// TwinCAT 3 PLC project Main
// ProgramVersion: 3.1.4023.0
// libraries:
//   Tc2_Standard, * (Beckhoff Automation GmbH)
//   Tc2_System, * (Beckhoff Automation GmbH)
//   Tc3_Module, * (Beckhoff Automation GmbH)
//   TcUnit, * (www.tcunit.org)
//   mobject-constants-datatype-limits,1.0.0,mobject
//   mobject-deserialization,0.3.0,mobject
//   mobject-errors,0.3.0,mobject
//   mobject-json,1.6.0,mobject
//   mobject-serialization,0.5.0,mobject
// project tree:
//   / PlcTask.TcTTO
//   POUs/ MAIN.TcPOU
//   Tests/ JsonDeserializerArrayForwardEnumerator_TestSuite.TcPOU, JsonDeserializerObjectForwardEnumerator_TestSuite.TcPOU, JsonDomParser_TestSuite.TcPOU, JsonSerializer_TestSuite.TcPOU, JsonDeserializer_TestSuite.TcPOU
//   Tests/Mocks/ MockSerializableUserObject.TcPOU, MockDeserializableUserObject.TcPOU, MockSerializableArray.TcPOU
// real-time tasks:
//   TASK PlcTask: cycle T#10ms, priority 20, ADS port 350

CONFIGURATION Main
    RESOURCE PLC ON TwinCAT3
        TASK PlcTask(INTERVAL := T#10ms, PRIORITY := 20);
        PROGRAM MAIN WITH PlcTask : MAIN;
    END_RESOURCE
END_CONFIGURATION

// ---- POUs/MAIN.TcPOU
PROGRAM MAIN
VAR
	jsonDomParser_TestSuite : JsonDomParser_TestSuite;
	jsonSerializer_TestSuite : JsonSerializer_TestSuite;
	jsonDeserializer_TestSuite : JsonDeserializer_TestSuite;
	jsonDeserializerArrayForwardEnumerator_TestSuite : JsonDeserializerArrayForwardEnumerator_TestSuite;
	jsonDeserializerObjectForwardEnumerator_TestSuite : JsonDeserializerObjectForwardEnumerator_TestSuite;
END_VAR

TcUnit.RUN();

END_PROGRAM

// ---- Tests/JsonDomParser_TestSuite.TcPOU
FUNCTION_BLOCK JsonDomParser_TestSuite EXTENDS TcUnit.FB_TestSuite
VAR
	jsonParser : JsonDomParser;
END_VAR

ModifyBoolArrayMemberFromJsonString();
ModifyDIntArrayMemberFromJsonString();
ModifyDIntPropertyFromJsonString();
ModifyFalseBoolPropertyFromJsonString();
ModifyIntArrayMemberFromJsonString();
ModifyIntPropertyFromJsonString();
ModifyLRealArrayMemberFromJsonString();
ModifyLRealPropertyFromJsonString();
ModifyRealArrayMemberFromJsonString();
ModifyRealPropertyFromJsonString();
ModifyStringPropertyFromJsonString();
ModifyTrueBoolPropertyFromJsonString();
ModifyUDIntArrayMemberFromJsonString();
ModifyUDIntPropertyFromJsonString();
ModifyValueFromChainedProperty();
ReadBoolArrayMemberFromJsonString();
ReadDIntArrayMemberFromJsonString();
ReadDIntPropertyFromJsonString();
ReadFalseBoolPropertyFromJsonString();
ReadIntArrayMemberFromJsonString();
ReadIntPropertyFromJsonString();
ReadLRealArrayMemberFromJsonString();
ReadLRealPropertyFromJsonString();
ReadRealArrayMemberFromJsonString();
ReadRealPropertyFromJsonString();
ReadStringPropertyFromJsonString();
ReadTrueBoolPropertyFromJsonString();
ReadUDIntArrayMemberFromJsonString();
ReadUDIntPropertyFromJsonString();
ReadValueFromChainedProperties();
TestTryLocateMethod();
TestTryWriteBoolMethod();
TestTryWriteDintMethod();
TestTryWriteIntMethod();
TestTryWriteLRealMethod();
TestTryWriteRealMethod();
TestTryWriteStringMethod();
TestTryWriteUdintMethod();

METHOD PUBLIC ModifyBoolArrayMemberFromJsonString
VAR_INPUT
END_VAR
VAR
	jsonTestString : T_MAXSTRING := '{"myArray" : [false, false, false]}';
	newValue : BOOL := TRUE;
	modifyResult : BOOL;
	result : BOOL;
	readResult : BOOL;
END_VAR
TEST('ModifyBoolArrayMemberFromJsonString');

// @TEST-RUN
jsonParser.ParseDocument(jsonTestString);
modifyResult := jsonParser.TryModify('.myArray[1]',newValue);
readResult := jsonParser.TryRead('.myArray[1]',result);
jsonParser.NewDocument();

// @TEST-ASSERT
AssertTrue(Condition := result, Message := 'Did not modify to the correct value');
AssertTrue(Condition := readResult, Message := 'Did not report a modify was successful');

TEST_FINISHED();
END_METHOD

METHOD PUBLIC ModifyDIntArrayMemberFromJsonString
VAR_INPUT
END_VAR
VAR
	jsonTestString : T_MAXSTRING := '{"myArray" : [123,456,789]}';
	newValue : DINT := 654;
	modifyResult : BOOL;
	actual : DINT;
	expected : DINT := 654;
	readResult : BOOL;
END_VAR
TEST('ModifyDIntArrayMemberFromJsonString');

// @TEST-RUN
jsonParser.ParseDocument(jsonTestString);
modifyResult := jsonParser.TryModify('.myArray[1]',newValue);
readResult := jsonParser.TryRead('.myArray[1]',actual);
jsonParser.NewDocument();

// @TEST-ASSERT
AssertEquals(Expected := expected, Actual := actual, Message := 'Did not modify to the correct value');
AssertTrue(Condition := modifyResult, Message := 'Did not report a modify was successful');

TEST_FINISHED();
END_METHOD

METHOD PUBLIC ModifyDIntPropertyFromJsonString
VAR_INPUT
END_VAR
VAR
	jsonTestString : T_MAXSTRING := '{"myDInt" : 123}';
	newValue : DINT := 456;
	modifyResult : BOOL;
	actual : DINT;
	expected : DINT := 456;
	readResult : BOOL;
END_VAR
TEST('ModifyDIntPropertyFromJsonString');

// @TEST-RUN
jsonParser.ParseDocument(jsonTestString);
modifyResult := jsonParser.TryModify('.myDInt',newValue);
readResult := jsonParser.TryRead('.myDInt',actual);
jsonParser.NewDocument();

// @TEST-ASSERT
AssertEquals(Expected := expected, Actual := actual, Message := 'Did not modify to the correct value');
AssertTrue(Condition := modifyResult, Message := 'Did not report a modify was successful');

TEST_FINISHED();
END_METHOD

METHOD PUBLIC ModifyFalseBoolPropertyFromJsonString
VAR_INPUT
END_VAR
VAR
	jsonTestString : T_MAXSTRING := '{"myTrueBool" : true, "myFalseBool" : false}';
	newValue : BOOL := TRUE;
	modifyResult : BOOL;
	result : BOOL;
	readResult : BOOL;
END_VAR
TEST('ModifyFalseBoolPropertyFromJsonString');

// @TEST-RUN
jsonParser.ParseDocument(jsonTestString);
modifyResult := jsonParser.TryModify('.myFalseBool',newValue);
readResult := jsonParser.TryRead('.myFalseBool',result);
jsonParser.NewDocument();

// @TEST-ASSERT
AssertTrue(Condition := result, Message := 'Did not modify to the correct value');
AssertTrue(Condition := modifyResult, Message := 'Did not report a modify was successful');

TEST_FINISHED();
END_METHOD

METHOD PUBLIC ModifyIntArrayMemberFromJsonString
VAR_INPUT
END_VAR
VAR
	jsonTestString : T_MAXSTRING := '{"myArray" : [123,456,789]}';
	newValue : INT := 654;
	modifyResult : BOOL;
	actual : INT;
	expected : INT := 654;
	readResult : BOOL;
END_VAR
TEST('ModifyIntArrayMemberFromJsonString');

// @TEST-RUN
jsonParser.ParseDocument(jsonTestString);
modifyResult := jsonParser.TryModify('.myArray[1]',newValue);
readResult := jsonParser.TryRead('.myArray[1]',actual);
jsonParser.NewDocument();

// @TEST-ASSERT
AssertEquals(Expected := expected, Actual := actual, Message := 'Did not modify to the correct value');
AssertTrue(Condition := modifyResult, Message := 'Did not report a modify was successful');

TEST_FINISHED();
END_METHOD

METHOD PUBLIC ModifyIntPropertyFromJsonString
VAR_INPUT
END_VAR
VAR
	jsonTestString : T_MAXSTRING := '{"myInt" : 123}';
	newValue : INT := 456;
	modifyResult : BOOL;
	actual : INT;
	expected : INT := 456;
	readResult : BOOL;
END_VAR
TEST('ModifyIntPropertyFromJsonString');

// @TEST-RUN
jsonParser.ParseDocument(jsonTestString);
modifyResult := jsonParser.TryModify('.myInt',newValue);
readResult := jsonParser.TryRead('.myInt',actual);
jsonParser.NewDocument();

// @TEST-ASSERT
AssertEquals(Expected := expected, Actual := actual, Message := 'Did not modify to the correct value');
AssertTrue(Condition := modifyResult, Message := 'Did not report a modify was successful');

TEST_FINISHED();
END_METHOD

METHOD PUBLIC ModifyLRealArrayMemberFromJsonString
VAR_INPUT
END_VAR
VAR
	jsonTestString : T_MAXSTRING := '{"myArray" : [123.1,456.2,789.3]}';
	newValue : LREAL := 678.4;
	modifyResult : BOOL;
	actual : LREAL;
	expected : LREAL := 678.4;
	readResult : BOOL;
END_VAR
TEST('ModifyLRealArrayMemberFromJsonString');

// @TEST-RUN
jsonParser.ParseDocument(jsonTestString);
modifyResult := jsonParser.TryModify('.myArray[1]',newValue);
readResult := jsonParser.TryRead('.myArray[1]',actual);
jsonParser.NewDocument();

// @TEST-ASSERT
AssertEquals(Expected := expected, Actual := actual, Message := 'Did not modify to the correct value');
AssertTrue(Condition := modifyResult, Message := 'Did not report a modify was successful');

TEST_FINISHED();
END_METHOD

METHOD PUBLIC ModifyLRealPropertyFromJsonString
VAR_INPUT
END_VAR
VAR
	jsonTestString : T_MAXSTRING := '{"myLReal" : 123.4}';
	newValue : LREAL := 456.5;
	modifyResult : BOOL;
	actual : LREAL;
	expected : LREAL := 456.5;
	readResult : BOOL;
END_VAR
TEST('ModifyLRealPropertyFromJsonString');

// @TEST-RUN
jsonParser.ParseDocument(jsonTestString);
modifyResult := jsonParser.TryModify('.myLReal',newValue);
readResult := jsonParser.TryRead('.myLReal',actual);
jsonParser.NewDocument();

// @TEST-ASSERT
AssertEquals(Expected := expected, Actual := actual, Message := 'Did not modify to the correct value');
AssertTrue(Condition := modifyResult, Message := 'Did not report a modify was successful');

TEST_FINISHED();
END_METHOD

METHOD PUBLIC ModifyRealArrayMemberFromJsonString
VAR_INPUT
END_VAR
VAR
	jsonTestString : T_MAXSTRING := '{"myArray" : [123.1,456.2,789.3]}';
	newValue : REAL := 678.4;
	modifyResult : BOOL;
	actual : REAL;
	expected : REAL := 678.4;
	readResult : BOOL;
END_VAR
TEST('ModifyRealArrayMemberFromJsonString');

// @TEST-RUN
jsonParser.ParseDocument(jsonTestString);
modifyResult := jsonParser.TryModify('.myArray[1]',newValue);
readResult := jsonParser.TryRead('.myArray[1]',actual);
jsonParser.NewDocument();

// @TEST-ASSERT
AssertEquals(Expected := expected, Actual := actual, Message := 'Did not modify to the correct value');
AssertTrue(Condition := modifyResult, Message := 'Did not report a modify was successful');

TEST_FINISHED();
END_METHOD

METHOD PUBLIC ModifyRealPropertyFromJsonString
VAR_INPUT
END_VAR
VAR
	jsonTestString : T_MAXSTRING := '{"myReal" : 123.4}';
	newValue : REAL := 456.5;
	modifyResult : BOOL;
	actual : REAL;
	expected : REAL := 456.5;
	readResult : BOOL;
END_VAR
TEST('ModifyRealPropertyFromJsonString');

// @TEST-RUN
jsonParser.ParseDocument(jsonTestString);
modifyResult := jsonParser.TryModify('.myReal',newValue);
readResult := jsonParser.TryRead('.myReal',actual);
jsonParser.NewDocument();

// @TEST-ASSERT
AssertEquals(Expected := expected, Actual := actual, Message := 'Did not modify to the correct value');
AssertTrue(Condition := modifyResult, Message := 'Did not report a modify was successful');

TEST_FINISHED();
END_METHOD

METHOD PUBLIC ModifyStringPropertyFromJsonString
VAR_INPUT
END_VAR
VAR
	jsonTestString : T_MAXSTRING := '{"myString" : "test"}';
	newValue : T_MAXSTRING := 'foobar';
	modifyResult : BOOL;
	actual : T_MAXSTRING;
	expected : T_MAXSTRING := 'foobar';
	readResult : BOOL;
END_VAR
TEST('ModifyStringPropertyFromJsonString');

// @TEST-RUN
jsonParser.ParseDocument(jsonTestString);
modifyResult := jsonParser.TryModify('.myString',newValue);
readResult := jsonParser.TryRead('.myString',actual);
jsonParser.NewDocument();

// @TEST-ASSERT
AssertEquals(Expected := expected, Actual := actual, Message := 'Did not modify to the correct value');
AssertTrue(Condition := modifyResult, Message := 'Did not report a modify was successful');

TEST_FINISHED();
END_METHOD

METHOD PUBLIC ModifyTrueBoolPropertyFromJsonString
VAR_INPUT
END_VAR
VAR
	jsonTestString : T_MAXSTRING := '{"myTrueBool" : true, "myFalseBool" : false}';
	newValue : BOOL := FALSE;
	modifyResult : BOOL;
	result : BOOL;
	readResult : BOOL;
END_VAR
TEST('ModifyTrueBoolPropertyFromJsonString');

// @TEST-RUN
jsonParser.ParseDocument(jsonTestString);
modifyResult := jsonParser.TryModify('.myTrueBool', newValue);
readResult := jsonParser.TryRead('.myTrueBool', result);
jsonParser.NewDocument();

// @TEST-ASSERT
AssertTrue(Condition := (result = newValue), Message := 'Did not modify to the correct value');
AssertTrue(Condition := modifyResult, Message := 'Did not report a modify was successful');

TEST_FINISHED();
END_METHOD

METHOD PUBLIC ModifyUDIntArrayMemberFromJsonString
VAR_INPUT
END_VAR
VAR
	jsonTestString : T_MAXSTRING := '{"myArray" : [123,456,789]}';
	newValue : UINT := 654;
	modifyResult : BOOL;
	actual : UINT;
	expected : UINT := 654;
	readResult : BOOL;
END_VAR
TEST('ModifyUDIntArrayMemberFromJsonString');

// @TEST-RUN
jsonParser.ParseDocument(jsonTestString);
modifyResult := jsonParser.TryModify('.myArray[1]',newValue);
readResult := jsonParser.TryRead('.myArray[1]',actual);
jsonParser.NewDocument();

// @TEST-ASSERT
AssertEquals(Expected := expected, Actual := actual, Message := 'Did not modify to the correct value');
AssertTrue(Condition := modifyResult, Message := 'Did not report a modify was successful');

TEST_FINISHED();
END_METHOD

METHOD PUBLIC ModifyUDIntPropertyFromJsonString
VAR_INPUT
END_VAR
VAR
	jsonTestString : T_MAXSTRING := '{"myUDInt" : 123}';
	newValue : UDINT := 456;
	modifyResult : BOOL;
	actual : UDINT;
	expected : UDINT := 456;
	readResult : BOOL;
END_VAR
TEST('ModifyUDIntPropertyFromJsonString');

// @TEST-RUN
jsonParser.ParseDocument(jsonTestString);
modifyResult := jsonParser.TryModify('.myUDInt',newValue);
readResult := jsonParser.TryRead('.myUDInt',actual);
jsonParser.NewDocument();

// @TEST-ASSERT
AssertEquals(Expected := expected, Actual := actual, Message := 'Did not modify to the correct value');
AssertTrue(Condition := modifyResult, Message := 'Did not report a modify was successful');

TEST_FINISHED();
END_METHOD

METHOD PUBLIC ModifyValueFromChainedProperty
VAR_INPUT
END_VAR
VAR
	jsonTestString : T_MAXSTRING := '{"level1" : {"level2" : {"level3" : {"level4" : 123}}}}';
	newValue : DINT := 456;
	modifyResult : BOOL;
	actual : DINT;
	expected : DINT := 456;
	readResult : BOOL;
END_VAR
TEST('ModifyValueFromChainedProperty');

// @TEST-RUN
jsonParser.ParseDocument(jsonTestString);
modifyResult := jsonParser.TryModify('.level1.level2.level3.level4',newValue);
readResult := jsonParser.TryRead('.level1.level2.level3.level4',actual);
jsonParser.NewDocument();

// @TEST-ASSERT
AssertEquals(Expected := expected, Actual := actual, Message := 'Did not modify to the correct value');
AssertTrue(Condition := modifyResult, Message := 'Did not report a modify was successful');

TEST_FINISHED();
END_METHOD

METHOD PUBLIC ReadBoolArrayMemberFromJsonString
VAR_INPUT
END_VAR
VAR
	jsonTestString : T_MAXSTRING := '{"myArray" : [false, true, false]}';
	result : BOOL;
	readResult : BOOL;
END_VAR
TEST('ReadBoolArrayMemberFromJsonString');

// @TEST-RUN
jsonParser.ParseDocument(jsonTestString);
readResult := jsonParser.TryRead('.myArray[1]',result);
jsonParser.NewDocument();

// @TEST-ASSERT
AssertTrue(Condition := result, Message := 'Did not read the correct value');
AssertTrue(Condition := readResult, Message := 'Did not report a read was successful');

TEST_FINISHED();
END_METHOD

METHOD PUBLIC ReadDIntArrayMemberFromJsonString
VAR_INPUT
END_VAR
VAR
	jsonTestString : T_MAXSTRING := '{"myArray" : [123,456,789]}';
	actual : DINT;
	expected : DINT := 456;
	readResult : BOOL;
END_VAR
TEST('ReadDIntArrayMemberFromJsonString');

// @TEST-RUN
jsonParser.ParseDocument(jsonTestString);
readResult := jsonParser.TryRead('.myArray[1]',Actual);
jsonParser.NewDocument();

// @TEST-ASSERT
AssertEquals(Expected := expected, Actual := actual, Message := 'Did not read the correct value');
AssertTrue(Condition := readResult, Message := 'Did not report a read was successful');

TEST_FINISHED();
END_METHOD

METHOD PUBLIC ReadDIntPropertyFromJsonString
VAR_INPUT
END_VAR
VAR
	jsonTestString : T_MAXSTRING := '{"myDInt" : 123}';
	actual : DINT;
	expected : DINT := 123;
	readResult : BOOL;
END_VAR
TEST('ReadDIntPropertyFromJsonString');

// @TEST-RUN
jsonParser.ParseDocument(jsonTestString);
readResult := jsonParser.TryRead('.myDInt',Actual);
jsonParser.NewDocument();

// @TEST-ASSERT
AssertEquals(Expected := expected, Actual := actual, Message := 'Did not read the correct value');
AssertTrue(Condition := readResult, Message := 'Did not report a read was successful');

TEST_FINISHED();
END_METHOD

METHOD PUBLIC ReadFalseBoolPropertyFromJsonString
VAR_INPUT
END_VAR
VAR
	jsonTestString : T_MAXSTRING := '{"myTrueBool" : true, "myFalseBool" : false}';
	result : BOOL;
	readResult : BOOL;
END_VAR
TEST('ReadFalseBoolPropertyFromJsonString');

// @TEST-RUN
jsonParser.ParseDocument(jsonTestString);
readResult := jsonParser.TryRead('.myFalseBool',result);
jsonParser.NewDocument();

// @TEST-ASSERT
AssertFalse(Condition := result, Message := 'Did not read the correct value');
AssertTrue(Condition := readResult, Message := 'Did not report a read was successful');

TEST_FINISHED();
END_METHOD

METHOD PUBLIC ReadIntArrayMemberFromJsonString
VAR_INPUT
END_VAR
VAR
	jsonTestString : T_MAXSTRING := '{"myArray" : [123,456,789]}';
	actual : INT;
	expected : INT := 456;
	readResult : BOOL;
END_VAR
TEST('ReadIntArrayMemberFromJsonString');

// @TEST-RUN
jsonParser.ParseDocument(jsonTestString);
readResult := jsonParser.TryRead('.myArray[1]',actual);
jsonParser.NewDocument();

// @TEST-ASSERT
AssertEquals(Expected := expected, Actual := actual, Message := 'Did not read the correct value');
AssertTrue(Condition := readResult, Message := 'Did not report a read was successful');

TEST_FINISHED();
END_METHOD

METHOD PUBLIC ReadIntPropertyFromJsonString
VAR_INPUT
END_VAR
VAR
	jsonTestString : T_MAXSTRING := '{"myInt" : 123}';
	actual : INT;
	expected : INT := 123;
	readResult : BOOL;
END_VAR
TEST('ReadIntPropertyFromJsonString');

// @TEST-RUN
jsonParser.ParseDocument(jsonTestString);
readResult := jsonParser.TryRead('.myInt',actual);
jsonParser.NewDocument();

// @TEST-ASSERT
AssertEquals(Expected := expected, Actual := actual, Message := 'Did not read the correct value');
AssertTrue(Condition := readResult, Message := 'Did not report a read was successful');

TEST_FINISHED();
END_METHOD

METHOD PUBLIC ReadLRealArrayMemberFromJsonString
VAR_INPUT
END_VAR
VAR
	jsonTestString : T_MAXSTRING := '{"myArray" : [-123.1,-456.2]}';
	actual : LREAL;
	expected : LREAL := -456.2;
	readResult : BOOL;
END_VAR
TEST('ReadLRealArrayMemberFromJsonString');

// @TEST-RUN
jsonParser.ParseDocument(jsonTestString);
readResult := jsonParser.TryRead('.myArray[1]',actual);
jsonParser.NewDocument();

// @TEST-ASSERT
AssertEquals(Expected := expected, Actual := actual, Message := 'Did not read the correct value');
AssertTrue(Condition := readResult, Message := 'Did not report a read was successful');

TEST_FINISHED();
END_METHOD

METHOD PUBLIC ReadLRealPropertyFromJsonString
VAR_INPUT
END_VAR
VAR
	jsonTestString : T_MAXSTRING := '{"myLReal" : -123.1}';
	actual : LREAL;
	expected : LREAL := -123.1;
	readResult : BOOL;
END_VAR
TEST('ReadLRealPropertyFromJsonString');

// @TEST-RUN
jsonParser.ParseDocument(jsonTestString);
readResult := jsonParser.TryRead('.myLReal',actual);
jsonParser.NewDocument();

// @TEST-ASSERT
AssertEquals(Expected := expected, Actual := actual, Message := 'Did not read the correct value');
AssertTrue(Condition := readResult, Message := 'Did not report a read was successful');

TEST_FINISHED();
END_METHOD

METHOD PUBLIC ReadRealArrayMemberFromJsonString
VAR_INPUT
END_VAR
VAR
	jsonTestString : T_MAXSTRING := '{"myArray" : [123.1,456.2,789.3]}';
	actual : REAL;
	expected : REAL := 456.2;
	readResult : BOOL;
END_VAR
TEST('ReadRealArrayMemberFromJsonString');

// @TEST-RUN
jsonParser.ParseDocument(jsonTestString);
readResult := jsonParser.TryRead('.myArray[1]',actual);
jsonParser.NewDocument();

// @TEST-ASSERT
AssertEquals(Expected := expected, Actual := actual, Message := 'Did not read the correct value');
AssertTrue(Condition := readResult, Message := 'Did not report a read was successful');

TEST_FINISHED();
END_METHOD

METHOD PUBLIC ReadRealPropertyFromJsonString
VAR_INPUT
END_VAR
VAR
	jsonTestString : T_MAXSTRING := '{"myReal" : 123.1}';
	actual : REAL;
	expected : REAL := 123.1;
	readResult : BOOL;
END_VAR
TEST('ReadRealPropertyFromJsonString');

// @TEST-RUN
jsonParser.ParseDocument(jsonTestString);
readResult := jsonParser.TryRead('.myReal',actual);
jsonParser.NewDocument();

// @TEST-ASSERT
AssertEquals(Expected := expected, Actual := actual, Message := 'Did not read the correct value');
AssertTrue(Condition := readResult, Message := 'Did not report a read was successful');

TEST_FINISHED();
END_METHOD

METHOD PUBLIC ReadStringPropertyFromJsonString
VAR_INPUT
END_VAR
VAR
	jsonTestString : T_MAXSTRING := '{"myString" : "test"}';
	actual : T_MAXSTRING;
	expected : T_MAXSTRING := 'test';
	readResult : BOOL;
END_VAR
TEST('ReadStringPropertyFromJsonString');

// @TEST-RUN
jsonParser.ParseDocument(jsonTestString);
readResult := jsonParser.TryRead('.myString',actual);
jsonParser.NewDocument();

// @TEST-ASSERT
AssertEquals(Expected := expected, Actual := actual, Message := 'Did not read the correct value');
AssertTrue(Condition := readResult, Message := 'Did not report a read was successful');

TEST_FINISHED();
END_METHOD

METHOD PUBLIC ReadTrueBoolPropertyFromJsonString
VAR_INPUT
END_VAR
VAR
	jsonTestString : T_MAXSTRING := '{"myTrueBool" : true, "myFalseBool" : false}';
	result : BOOL;
	readResult : BOOL;
END_VAR
TEST('ReadTrueBoolPropertyFromJsonString');

// @TEST-RUN
jsonParser.ParseDocument(jsonTestString);
readResult := jsonParser.TryRead('.myTrueBool',result);
jsonParser.NewDocument();

// @TEST-ASSERT
AssertTrue(Condition := result, Message := 'Did not read the correct value');
AssertTrue(Condition := readResult, Message := 'Did not report a read was successful');

TEST_FINISHED();
END_METHOD

METHOD PUBLIC ReadUDIntArrayMemberFromJsonString
VAR_INPUT
END_VAR
VAR
	jsonTestString : T_MAXSTRING := '{"myArray" : [123,456,789]}';
	actual : UDINT;
	expected : UDINT := 456;
	readResult : BOOL;
END_VAR
TEST('ReadUDIntArrayMemberFromJsonString');

// @TEST-RUN
jsonParser.ParseDocument(jsonTestString);
readResult := jsonParser.TryRead('.myArray[1]',actual);
jsonParser.NewDocument();

// @TEST-ASSERT
AssertEquals(Expected := expected, Actual := actual, Message := 'Did not read the correct value');
AssertTrue(Condition := readResult, Message := 'Did not report a read was successful');

TEST_FINISHED();
END_METHOD

METHOD PUBLIC ReadUDIntPropertyFromJsonString
VAR_INPUT
END_VAR
VAR
	jsonTestString : T_MAXSTRING := '{"myUDInt" : 123}';
	actual : UDINT;
	expected : UDINT := 123;
	readResult : BOOL;
END_VAR
TEST('ReadUDIntPropertyFromJsonString');

// @TEST-RUN
jsonParser.ParseDocument(jsonTestString);
readResult := jsonParser.TryRead('.myUDInt',actual);
jsonParser.NewDocument();

// @TEST-ASSERT
AssertEquals(Expected := expected, Actual := actual, Message := 'Did not read the correct value');
AssertTrue(Condition := readResult, Message := 'Did not report a read was successful');

TEST_FINISHED();
END_METHOD

METHOD PUBLIC ReadValueFromChainedProperties
VAR_INPUT
END_VAR
VAR
	jsonTestString : T_MAXSTRING := '{"level1" : {"level2" : {"level3" : {"level4" : 123}}}}';
	actual : DINT;
	expected : DINT := 123;
	readResult : BOOL;
END_VAR
TEST('ReadValueFromChainedProperties');

// @TEST-RUN
jsonParser.ParseDocument(jsonTestString);
readResult := jsonParser.TryRead('.level1.level2.level3.level4',actual);
jsonParser.NewDocument();

// @TEST-ASSERT
AssertEquals(Expected := expected, Actual := actual, Message := 'Did not read the correct value');
AssertTrue(Condition := readResult, Message := 'Did not report a read was successful');

TEST_FINISHED();
END_METHOD

METHOD PUBLIC TestTryLocateMethod
VAR_INPUT
END_VAR
VAR
	jsonTestString : T_MAXSTRING := '{"level1" : {"level2" : "test"}}';
	root : SJsonValue;
	level1 : SJsonValue;
	level2 : SJsonValue;
	actual : SJsonValue;
	locateResult : BOOL;
END_VAR
TEST('TestTryLocateMethod');

// @TEST-RUN
root := jsonParser.ParseDocument(jsonTestString);

// manually obtain the correct result
level1 := jsonParser.FindMember(root,'level1');
level2 := jsonParser.FindMember(level1,'level2');

locateResult := jsonParser.TryLocate('.level1.level2',actual);
jsonParser.NewDocument();

// @TEST-ASSERT
AssertEquals(Expected := level2, Actual := actual, Message := 'Did not locate the correct member');
AssertTrue(Condition := locateResult, Message := 'Did not report a locate was successful');

TEST_FINISHED();
END_METHOD

METHOD TestTryWriteBoolMethod
VAR
    jsonParser : JsonDomParser;
    jsonInitialString : T_MAXSTRING := '{"foo":"bar"}';
    newBool : BOOL := TRUE;  // Example BOOL value
    writeSuccess1 : BOOL;
    writeSuccess2 : BOOL;
    readBool1 : BOOL;
    readBool2 : BOOL;
    readResult1 : BOOL;
    readResult2 : BOOL;
    jsonOutput : T_MAXSTRING;
    expectedJsonOutput : T_MAXSTRING := '{"foo":"bar","myThing":[null,null,{"myBoolValue":true},null,true]}';
END_VAR
TEST('TestTryWriteBOOLMethod');

// @TEST-RUN
jsonParser.ParseDocument(jsonInitialString);
writeSuccess1 := jsonParser.TryWrite('.myThing[2].myBoolValue', newBool);
writeSuccess2 := jsonParser.TryWrite('.myThing[4]', newBool);
jsonOutput := jsonParser.GetDocument();

readResult1 := jsonParser.TryRead('.myThing[2].myBoolValue', readBool1);
readResult2 := jsonParser.TryRead('.myThing[4]', readBool2);
jsonParser.NewDocument();

// @TEST-ASSERT
AssertTrue(Condition := writeSuccess1, Message := 'First TryWrite operation was unsuccessful for BOOL');
AssertTrue(Condition := writeSuccess2, Message := 'Second TryWrite operation was unsuccessful for BOOL');
AssertTrue(Condition := readResult1 AND (readBool1 = newBool), Message := 'Could not read back the first written BOOL value or value mismatched');
AssertTrue(Condition := readResult2 AND (readBool2 = newBool), Message := 'Could not read back the second written BOOL value or value mismatched');
AssertEquals(Expected := expectedJsonOutput, Actual := jsonOutput, Message := 'Output JSON does not match expected for BOOL');

TEST_FINISHED();
END_METHOD

METHOD TestTryWriteDintMethod
VAR
    jsonParser : JsonDomParser;
    jsonInitialString : T_MAXSTRING := '{"foo":"bar"}';
    newDInt : DINT := -12345678;  // Example DINT value (can be negative)
    writeSuccess1 : BOOL;
    writeSuccess2 : BOOL;
    readDInt1 : DINT;
    readDInt2 : DINT;
    readResult1 : BOOL;
    readResult2 : BOOL;
    jsonOutput : T_MAXSTRING;
    expectedJsonOutput : T_MAXSTRING := '{"foo":"bar","myThing":[null,null,{"myDIntValue":-12345678},null,-12345678]}';
END_VAR
TEST('TestTryWriteDINTMethod');

// @TEST-RUN
jsonParser.ParseDocument(jsonInitialString);
writeSuccess1 := jsonParser.TryWrite('.myThing[2].myDIntValue', newDInt);
writeSuccess2 := jsonParser.TryWrite('.myThing[4]', newDInt);
jsonOutput := jsonParser.GetDocument();

readResult1 := jsonParser.TryRead('.myThing[2].myDIntValue', readDInt1);
readResult2 := jsonParser.TryRead('.myThing[4]', readDInt2);
jsonParser.NewDocument();

// @TEST-ASSERT
AssertTrue(Condition := writeSuccess1, Message := 'First TryWrite operation was unsuccessful for DINT');
AssertTrue(Condition := writeSuccess2, Message := 'Second TryWrite operation was unsuccessful for DINT');
AssertTrue(Condition := readResult1 AND (readDInt1 = newDInt), Message := 'Could not read back the first written DINT value or value mismatched');
AssertTrue(Condition := readResult2 AND (readDInt2 = newDInt), Message := 'Could not read back the second written DINT value or value mismatched');
AssertEquals(Expected := expectedJsonOutput, Actual := jsonOutput, Message := 'Output JSON does not match expected for DINT');

TEST_FINISHED();
END_METHOD

METHOD TestTryWriteIntMethod
VAR
    jsonParser : JsonDomParser;
    jsonInitialString : T_MAXSTRING := '{"foo":"bar"}';
    newInt : INT := 789;
    writeSuccess1 : BOOL;
    writeSuccess2 : BOOL;
    readInt1 : INT;
    readInt2 : INT;
    readResult1 : BOOL;
    readResult2 : BOOL;
    jsonOutput : T_MAXSTRING;
    expectedJsonOutput : T_MAXSTRING := '{"foo":"bar","myThing":[null,null,{"myIntValue":789},null,789]}';
END_VAR
TEST('TestTryWriteIntMethod');

// @TEST-RUN
jsonParser.ParseDocument(jsonInitialString);
writeSuccess1 := jsonParser.TryWrite('.myThing[2].myIntValue', newInt);
writeSuccess2 := jsonParser.TryWrite('.myThing[4]', newInt);
jsonOutput := jsonParser.GetDocument();

readResult1 := jsonParser.TryRead('.myThing[2].myIntValue', readInt1);
readResult2 := jsonParser.TryRead('.myThing[4]', readInt2);
jsonParser.NewDocument();

// @TEST-ASSERT
AssertTrue(Condition := writeSuccess1, Message := 'First TryWrite operation was unsuccessful');
AssertTrue(Condition := writeSuccess2, Message := 'Second TryWrite operation was unsuccessful');
AssertTrue(Condition := readResult1 AND (readInt1 = newInt), Message := 'Could not read back the first written INT value or value mismatched');
AssertTrue(Condition := readResult2 AND (readInt2 = newInt), Message := 'Could not read back the second written INT value or value mismatched');
AssertEquals(Expected := expectedJsonOutput, Actual := jsonOutput, Message := 'Output JSON does not match expected');

TEST_FINISHED();
END_METHOD

METHOD TestTryWriteLRealMethod
VAR
    jsonParser : JsonDomParser;
    jsonInitialString : T_MAXSTRING := '{"foo":"bar"}';
    newLReal : LREAL := 12345.6789;  // Example LREAL value
    writeSuccess1 : BOOL;
    writeSuccess2 : BOOL;
    readLReal1 : LREAL;
    readLReal2 : LREAL;
    readResult1 : BOOL;
    readResult2 : BOOL;
    jsonOutput : T_MAXSTRING;
    expectedJsonOutput : T_MAXSTRING := '{"foo":"bar","myThing":[null,null,{"myLRealValue":12345.6789},null,12345.6789]}';
END_VAR
TEST('TestTryWriteLREALMethod');

// @TEST-RUN
jsonParser.ParseDocument(jsonInitialString);
writeSuccess1 := jsonParser.TryWrite('.myThing[2].myLRealValue', newLReal);
writeSuccess2 := jsonParser.TryWrite('.myThing[4]', newLReal);
jsonOutput := jsonParser.GetDocument();

readResult1 := jsonParser.TryRead('.myThing[2].myLRealValue', readLReal1);
readResult2 := jsonParser.TryRead('.myThing[4]', readLReal2);
jsonParser.NewDocument();

// @TEST-ASSERT
AssertTrue(Condition := writeSuccess1, Message := 'First TryWrite operation was unsuccessful for LREAL');
AssertTrue(Condition := writeSuccess2, Message := 'Second TryWrite operation was unsuccessful for LREAL');
AssertTrue(Condition := readResult1 AND ABS(readLReal1 - newLReal) < 1e-6, Message := 'Could not read back the first written LREAL value or value mismatched');  // using a tolerance for floating-point comparison
AssertTrue(Condition := readResult2 AND ABS(readLReal2 - newLReal) < 1e-6, Message := 'Could not read back the second written LREAL value or value mismatched');  // using a tolerance for floating-point comparison
AssertEquals(Expected := expectedJsonOutput, Actual := jsonOutput, Message := 'Output JSON does not match expected for LREAL');

TEST_FINISHED();
END_METHOD

METHOD TestTryWriteRealMethod
VAR
    jsonParser : JsonDomParser;
    jsonInitialString : T_MAXSTRING := '{"foo":"bar"}';
    newReal : REAL := 123.456;  // Example REAL value
    writeSuccess1 : BOOL;
    writeSuccess2 : BOOL;
    readReal1 : REAL;
    readReal2 : REAL;
    readResult1 : BOOL;
    readResult2 : BOOL;
    jsonOutput : T_MAXSTRING;
    expectedJsonOutput : T_MAXSTRING := '{"foo":"bar","myThing":[null,null,{"myRealValue":123.456},null,123.456]}';
END_VAR
TEST('TestTryWriteREALMethod');

// @TEST-RUN
jsonParser.ParseDocument(jsonInitialString);
writeSuccess1 := jsonParser.TryWrite('.myThing[2].myRealValue', newReal);
writeSuccess2 := jsonParser.TryWrite('.myThing[4]', newReal);
jsonOutput := jsonParser.GetDocument();

readResult1 := jsonParser.TryRead('.myThing[2].myRealValue', readReal1);
readResult2 := jsonParser.TryRead('.myThing[4]', readReal2);
jsonParser.NewDocument();

// @TEST-ASSERT
AssertTrue(Condition := writeSuccess1, Message := 'First TryWrite operation was unsuccessful for REAL');
AssertTrue(Condition := writeSuccess2, Message := 'Second TryWrite operation was unsuccessful for REAL');
AssertTrue(Condition := readResult1 AND ABS(readReal1 - newReal) < 1e-5, Message := 'Could not read back the first written REAL value or value mismatched');  // using a tolerance for floating-point comparison
AssertTrue(Condition := readResult2 AND ABS(readReal2 - newReal) < 1e-5, Message := 'Could not read back the second written REAL value or value mismatched');  // using a tolerance for floating-point comparison
//AssertEquals(Expected := expectedJsonOutput, Actual := jsonOutput, Message := 'Output JSON does not match expected for REAL');

TEST_FINISHED();
END_METHOD

METHOD TestTryWriteStringMethod
VAR
    jsonParser : JsonDomParser;
    jsonInitialString : T_MAXSTRING := '{"foo":"bar"}';
    newString : STRING := 'HelloWorld';  // Example STRING value
    writeSuccess1 : BOOL;
    writeSuccess2 : BOOL;
    readString1 : STRING;
    readString2 : STRING;
    readResult1 : BOOL;
    readResult2 : BOOL;
    jsonOutput : T_MAXSTRING;
    expectedJsonOutput : T_MAXSTRING := '{"foo":"bar","myThing":[null,null,{"myStringValue":"HelloWorld"},null,"HelloWorld"]}';
END_VAR
TEST('TestTryWriteSTRINGMethod');

// @TEST-RUN
jsonParser.ParseDocument(jsonInitialString);
writeSuccess1 := jsonParser.TryWrite('.myThing[2].myStringValue', newString);
writeSuccess2 := jsonParser.TryWrite('.myThing[4]', newString);
jsonOutput := jsonParser.GetDocument();

readResult1 := jsonParser.TryRead('.myThing[2].myStringValue', readString1);
readResult2 := jsonParser.TryRead('.myThing[4]', readString2);
jsonParser.NewDocument();

// @TEST-ASSERT
AssertTrue(Condition := writeSuccess1, Message := 'First TryWrite operation was unsuccessful for STRING');
AssertTrue(Condition := writeSuccess2, Message := 'Second TryWrite operation was unsuccessful for STRING');
AssertTrue(Condition := readResult1 AND (readString1 = newString), Message := 'Could not read back the first written STRING value or value mismatched');
AssertTrue(Condition := readResult2 AND (readString2 = newString), Message := 'Could not read back the second written STRING value or value mismatched');
AssertEquals(Expected := expectedJsonOutput, Actual := jsonOutput, Message := 'Output JSON does not match expected for STRING');

TEST_FINISHED();
END_METHOD

METHOD TestTryWriteUdintMethod
VAR
    jsonParser : JsonDomParser;
    jsonInitialString : T_MAXSTRING := '{"foo":"bar"}';
    newUDInt : UDINT := 1234567890;  // Assuming UDINT has a suitable range
    writeSuccess1 : BOOL;
    writeSuccess2 : BOOL;
    readUDInt1 : UDINT;
    readUDInt2 : UDINT;
    readResult1 : BOOL;
    readResult2 : BOOL;
    jsonOutput : T_MAXSTRING;
    expectedJsonOutput : T_MAXSTRING := '{"foo":"bar","myThing":[null,null,{"myUDIntValue":1234567890},null,1234567890]}';
END_VAR
TEST('TestTryWriteUDINTMethod');

// @TEST-RUN
jsonParser.ParseDocument(jsonInitialString);
writeSuccess1 := jsonParser.TryWrite('.myThing[2].myUDIntValue', newUDInt);
writeSuccess2 := jsonParser.TryWrite('.myThing[4]', newUDInt);
jsonOutput := jsonParser.GetDocument();

readResult1 := jsonParser.TryRead('.myThing[2].myUDIntValue', readUDInt1);
readResult2 := jsonParser.TryRead('.myThing[4]', readUDInt2);
jsonParser.NewDocument();

// @TEST-ASSERT
AssertTrue(Condition := writeSuccess1, Message := 'First TryWrite operation was unsuccessful for UDINT');
AssertTrue(Condition := writeSuccess2, Message := 'Second TryWrite operation was unsuccessful for UDINT');
AssertTrue(Condition := readResult1 AND (readUDInt1 = newUDInt), Message := 'Could not read back the first written UDINT value or value mismatched');
AssertTrue(Condition := readResult2 AND (readUDInt2 = newUDInt), Message := 'Could not read back the second written UDINT value or value mismatched');
AssertEquals(Expected := expectedJsonOutput, Actual := jsonOutput, Message := 'Output JSON does not match expected for UDINT');

TEST_FINISHED();
END_METHOD

END_FUNCTION_BLOCK

// ---- Tests/JsonSerializer_TestSuite.TcPOU
FUNCTION_BLOCK JsonSerializer_TestSuite EXTENDS TcUnit.FB_TestSuite

TestAddBase64();
TestAddBoolWithFalseBoolVariable();
TestAddBoolWithTrueBoolVariable();
TestAddByte();
TestAddBytesAsHex();
TestAddDateTime();
TestAddDcTime();
TestAddDint();
TestAddDword();
TestAddFileTime();
TestAddInt();
TestAddKey();
TestAddKeyBase64();
TestAddKeyBoolWithFalseBoolVariable();
TestAddKeyBoolWithTrueBoolVariable();
TestAddKeyByte();
TestAddKeyBytesAsHex();
TestAddKeyDateTime();
TestAddKeyDcTime();
TestAddKeyDint();
TestAddKeyDword();
TestAddKeyFileTime();
TestAddKeyInt();
TestAddKeyLint();
TestAddKeyLreal();
TestAddKeyLreal_Max();
TestAddKeyLtime();
TestAddKeyLword();
TestAddKeyNull();
TestAddKeyObject();
TestAddKeyObject_Array();
TestAddKeyRawJson();
TestAddKeyReal();
TestAddKeyReal_Max();
TestAddKeySint();
TestAddKeyString();
TestAddKeyStringByRef();
TestAddKeyTime();
TestAddKeyTod();
TestAddKeyUdint();
TestAddKeyUint();
TestAddKeyUlint();
TestAddKeyUsint();
TestAddKeyWord();
TestAddLint();
TestAddLreal();
TestAddLtime();
TestAddLword();
TestAddNull();
TestAddObject();
TestAddObjects();
TestAddRawJson();
TestAddReal();
TestAddSint();
TestAddString();
TestAddStringByRef();
TestAddTime();
TestAddTod();
TestAddUdint();
TestAddUint();
TestAddUlint();
TestAddUsint();
TestAddWord();
TestClone();
TestGetSerializedDataLengthEmpty();
TestGetSerializedDataLengthWithEmptyObject();
TestGetSerializedDataLengthWithSimpleObject();
TestReset();
TestSerializeArray();
TestSerializeObject();

METHOD PUBLIC TestAddBase64
VAR
	jsonSerializer : JsonSerializer;
	rawData : ARRAY[0..4] OF BYTE := [104, 101, 108, 108, 111];
	out : STRING;
	expected : STRING := '"aGVsbG8="';
END_VAR
TEST('TestAddBase64');

jsonSerializer.AddBase64(ADR(rawData), SIZEOF(rawData));
jsonSerializer.TryGetSerializedData(ADR(out),SIZEOF(out));

AssertEquals(
	Expected := expected,
	Actual := out,
	Message := 'Did not produce the expected JSON string for Base64 encoded "hello"'
);

TEST_FINISHED();
END_METHOD

METHOD PUBLIC TestAddBoolWithFalseBoolVariable
VAR
	jsonSerializer : JsonSerializer;
	value : BOOL := FALSE;
	out : STRING;
	expected : STRING := 'false';
END_VAR
TEST('TestAddBoolWithFalseBoolVariable');

jsonSerializer.AddBool(value);
jsonSerializer.TryGetSerializedData(ADR(out),SIZEOF(out));

AssertEquals(
	Expected := expected,
	Actual := out,
	Message := 'Did not produce the expected JSON string for a false value'
);

TEST_FINISHED();
END_METHOD

METHOD PUBLIC TestAddBoolWithTrueBoolVariable
VAR
	jsonSerializer : JsonSerializer;
	value : BOOL := TRUE;
	out : STRING;
	expected : STRING := 'true';
END_VAR
TEST('TestAddBoolWithTrueBoolVariable');

jsonSerializer.AddBool(value);
jsonSerializer.TryGetSerializedData(ADR(out),SIZEOF(out));

AssertEquals(
	Expected := expected,
	Actual := out,
	Message := 'Did not produce the expected JSON string for a true value'
);

TEST_FINISHED();
END_METHOD

METHOD PUBLIC TestAddByte
VAR
	jsonSerializer : JsonSerializer;
	byteValue : BYTE := 100;
	out : STRING;
	expected : STRING := '100';
END_VAR
TEST('TestAddByte');

jsonSerializer.AddByte(byteValue);
jsonSerializer.TryGetSerializedData(ADR(out),SIZEOF(out));

AssertEquals(
	Expected := expected,
	Actual := out,
	Message := 'Did not produce the expected JSON string for the BYTE value'
);

TEST_FINISHED();
END_METHOD

METHOD PUBLIC TestAddBytesAsHex
VAR
	jsonSerializer : JsonSerializer;
	binaryData : ARRAY[0..3] OF BYTE := [16#BA, 16#AD, 16#F0, 16#0D];
	out : STRING;
	expected : STRING := '"baadf00d"';
END_VAR
TEST('TestAddBytesAsHex');

jsonSerializer.AddBytesAsHex(ADR(binaryData), SIZEOF(binaryData));
jsonSerializer.TryGetSerializedData(ADR(out),SIZEOF(out));

AssertEquals(
	Expected := expected,
	Actual := out,
	Message := 'Did not produce the expected JSON string for hexadecimal binary data'
);

TEST_FINISHED();
END_METHOD

METHOD PUBLIC TestAddDateTime
VAR
	jsonSerializer : JsonSerializer;
	dateTimeValue : DATE_AND_TIME := DT#2023-12-30-15:20:00;
	out : STRING;
	expected : STRING := '"2023-12-30T15:20:00"';
END_VAR
TEST('TestAddDateTime');

jsonSerializer.AddDateTime(dateTimeValue);
jsonSerializer.TryGetSerializedData(ADR(out),SIZEOF(out));

AssertEquals(
	Expected := expected,
	Actual := out,
	Message := 'Did not produce the expected JSON string for the DATE_AND_TIME value'
);

TEST_FINISHED();
END_METHOD

METHOD PUBLIC TestAddDcTime
VAR
	jsonSerializer : JsonSerializer;
	dcTimeValue : DCTIME := 12345678;
	out : STRING;
	expected : STRING := '"2000-01-01T00:00:00.012345678"';
END_VAR
TEST('TestAddDcTime');

jsonSerializer.AddDcTime(dcTimeValue);
jsonSerializer.TryGetSerializedData(ADR(out),SIZEOF(out));

AssertEquals(
	Expected := expected,
	Actual := out,
	Message := 'Did not produce the expected JSON string for the DCTIME value'
);

TEST_FINISHED();
END_METHOD

METHOD PUBLIC TestAddDint
VAR
	jsonSerializer : JsonSerializer;
	dintValue : DINT := 12345;
	out : STRING;
	expected : STRING := '12345';
END_VAR
TEST('TestAddDint');

jsonSerializer.AddDint(dintValue);
jsonSerializer.TryGetSerializedData(ADR(out),SIZEOF(out));

AssertEquals(
	Expected := expected,
	Actual := out,
	Message := 'Did not produce the expected JSON string for the DINT value'
);

TEST_FINISHED();
END_METHOD

METHOD PUBLIC TestAddDword
VAR
	jsonSerializer : JsonSerializer;
	dwordValue : DWORD := 12345;
	out : STRING;
	expected : STRING := '12345';
END_VAR
TEST('TestAddDword');

jsonSerializer.AddDword(dwordValue);
jsonSerializer.TryGetSerializedData(ADR(out),SIZEOF(out));

AssertEquals(
	Expected := expected,
	Actual := out,
	Message := 'Did not produce the expected JSON string for the DWORD value'
);

TEST_FINISHED();
END_METHOD

METHOD PUBLIC TestAddFileTime
VAR
	jsonSerializer : JsonSerializer;
	fileTimeValue : FILETIME := 12345678;
	out : STRING;
	expected : STRING := '"1601-01-01T00:00:01.2345678"';
END_VAR
TEST('TestAddFileTime');

jsonSerializer.AddFileTime(fileTimeValue);
jsonSerializer.TryGetSerializedData(ADR(out),SIZEOF(out));

AssertEquals(
	Expected := expected,
	Actual := out,
	Message := 'Did not produce the expected JSON string for the FileTime value'
);

TEST_FINISHED();
END_METHOD

METHOD PUBLIC TestAddInt
VAR
	jsonSerializer : JsonSerializer;
	intValue : INT := 12345;
	out : STRING;
	expected : STRING := '12345';
END_VAR
TEST('TestAddInt');

jsonSerializer.AddInt(intValue);
jsonSerializer.TryGetSerializedData(ADR(out),SIZEOF(out));

AssertEquals(
	Expected := expected,
	Actual := out,
	Message := 'Did not produce the expected JSON string for the INT value'
);

TEST_FINISHED();
END_METHOD

METHOD PUBLIC TestAddKey
VAR
	jsonSerializer : JsonSerializer;
	out : STRING;
	expected : STRING := '{"data":123}';
END_VAR
TEST('TestAddKey');

jsonSerializer.StartObject();
jsonSerializer.AddKey('data');
jsonSerializer.AddDint(123);
jsonSerializer.EndObject();

jsonSerializer.TryGetSerializedData(ADR(out),SIZEOF(out));

AssertEquals(
	Expected := expected,
	Actual := out,
	Message := 'Did not produce the expected JSON string for the KEY value'
);

TEST_FINISHED();
END_METHOD

METHOD PUBLIC TestAddKeyBase64
VAR
	jsonSerializer : JsonSerializer;
	rawData : ARRAY[0..4] OF BYTE := [104, 101, 108, 108, 111];
	out : STRING;
	expected : STRING := '{"data":"aGVsbG8="}';
END_VAR
TEST('TestAddKeyBase64');

jsonSerializer.StartObject();
jsonSerializer.AddKeyBase64('data',ADR(rawData), SIZEOF(rawData));
jsonSerializer.EndObject();

jsonSerializer.TryGetSerializedData(ADR(out),SIZEOF(out));

AssertEquals(
	Expected := expected,
	Actual := out,
	Message := 'Did not produce the expected JSON string for Base64 encoded "hello"'
);

TEST_FINISHED();
END_METHOD

METHOD PUBLIC TestAddKeyBoolWithFalseBoolVariable
VAR
	jsonSerializer : JsonSerializer;
	value : BOOL := FALSE;
	out : STRING;
	expected : STRING := '{"data":false}';
END_VAR
TEST('TestAddKeyBoolWithFalseBoolVariable');

jsonSerializer.StartObject();
jsonSerializer.AddKeyBool('data',value);
jsonSerializer.EndObject();

jsonSerializer.TryGetSerializedData(ADR(out),SIZEOF(out));

AssertEquals(
	Expected := expected,
	Actual := out,
	Message := 'Did not produce the expected JSON string for a false value'
);

TEST_FINISHED();
END_METHOD

METHOD PUBLIC TestAddKeyBoolWithTrueBoolVariable
VAR
	jsonSerializer : JsonSerializer;
	value : BOOL := TRUE;
	out : STRING;
	expected : STRING := '{"data":true}';
END_VAR
TEST('TestAddKeyBoolWithTrueBoolVariable');

jsonSerializer.StartObject();
jsonSerializer.AddKeyBool('data',value);
jsonSerializer.EndObject();

jsonSerializer.TryGetSerializedData(ADR(out),SIZEOF(out));

AssertEquals(
	Expected := expected,
	Actual := out,
	Message := 'Did not produce the expected JSON string for a true value'
);

TEST_FINISHED();
END_METHOD

METHOD PUBLIC TestAddKeyByte
VAR
	jsonSerializer : JsonSerializer;
	byteValue : BYTE := 100;
	out : STRING;
	expected : STRING := '{"data":100}';
END_VAR
TEST('TestAddKeyByte');

jsonSerializer.StartObject();
jsonSerializer.AddKeyByte('data',byteValue);
jsonSerializer.EndObject();

jsonSerializer.TryGetSerializedData(ADR(out),SIZEOF(out));

AssertEquals(
	Expected := expected,
	Actual := out,
	Message := 'Did not produce the expected JSON string for the BYTE value'
);

TEST_FINISHED();
END_METHOD

METHOD PUBLIC TestAddKeyBytesAsHex
VAR
	jsonSerializer : JsonSerializer;
	binaryData : ARRAY[0..3] OF BYTE := [16#BA, 16#AD, 16#F0, 16#0D];
	out : STRING;
	expected : STRING := '{"data":"baadf00d"}';
END_VAR
TEST('TestAddKeyBytesAsHex');

jsonSerializer.StartObject();
jsonSerializer.AddKeyBytesAsHex('data',ADR(binaryData), SIZEOF(binaryData));
jsonSerializer.EndObject();

jsonSerializer.TryGetSerializedData(ADR(out),SIZEOF(out));

AssertEquals(
	Expected := expected,
	Actual := out,
	Message := 'Did not produce the expected JSON string for hexadecimal binary data'
);

TEST_FINISHED();
END_METHOD

METHOD PUBLIC TestAddKeyDateTime
VAR
	jsonSerializer : JsonSerializer;
	dateTimeValue : DATE_AND_TIME := DT#2023-12-30-15:20:00;
	out : STRING;
	expected : STRING := '{"data":"2023-12-30T15:20:00"}';
END_VAR
TEST('TestAddKeyDateTime');

jsonSerializer.StartObject();
jsonSerializer.AddKeyDateTime('data',dateTimeValue);
jsonSerializer.EndObject();

jsonSerializer.TryGetSerializedData(ADR(out),SIZEOF(out));

AssertEquals(
	Expected := expected,
	Actual := out,
	Message := 'Did not produce the expected JSON string for the DATE_AND_TIME value'
);

TEST_FINISHED();
END_METHOD

METHOD PUBLIC TestAddKeyDcTime
VAR
	jsonSerializer : JsonSerializer;
	dcTimeValue : DCTIME := 12345678;
	out : STRING;
	expected : STRING := '{"data":"2000-01-01T00:00:00.012345678"}';
END_VAR
TEST('TestAddKeyDcTime');

jsonSerializer.StartObject();
jsonSerializer.AddKeyDcTime('data',dcTimeValue);
jsonSerializer.EndObject();

jsonSerializer.TryGetSerializedData(ADR(out),SIZEOF(out));

AssertEquals(
	Expected := expected,
	Actual := out,
	Message := 'Did not produce the expected JSON string for the DCTIME value'
);

TEST_FINISHED();
END_METHOD

METHOD PUBLIC TestAddKeyDint
VAR
	jsonSerializer : JsonSerializer;
	dintValue : DINT := 12345;
	out : STRING;
	expected : STRING := '{"data":12345}';
END_VAR
TEST('TestAddKeyDint');

jsonSerializer.StartObject();
jsonSerializer.AddKeyDint('data',dintValue);
jsonSerializer.EndObject();

jsonSerializer.TryGetSerializedData(ADR(out),SIZEOF(out));

AssertEquals(
	Expected := expected,
	Actual := out,
	Message := 'Did not produce the expected JSON string for the DINT value'
);

TEST_FINISHED();
END_METHOD

METHOD PUBLIC TestAddKeyDword
VAR
	jsonSerializer : JsonSerializer;
	dwordValue : DWORD := 12345;
	out : STRING;
	expected : STRING := '{"data":12345}';
END_VAR
TEST('TestAddKeyDword');

jsonSerializer.StartObject();
jsonSerializer.AddKeyDword('data',dwordValue);
jsonSerializer.EndObject();

jsonSerializer.TryGetSerializedData(ADR(out),SIZEOF(out));

AssertEquals(
	Expected := expected,
	Actual := out,
	Message := 'Did not produce the expected JSON string for the DWORD value'
);

TEST_FINISHED();
END_METHOD

METHOD PUBLIC TestAddKeyFileTime
VAR
	jsonSerializer : JsonSerializer;
	fileTimeValue : FILETIME := 12345678;
	out : STRING;
	expected : STRING := '{"data":"1601-01-01T00:00:01.2345678"}';
END_VAR
TEST('TestAddKeyFileTime');

jsonSerializer.StartObject();
jsonSerializer.AddKeyFileTime('data',fileTimeValue);
jsonSerializer.EndObject();

jsonSerializer.TryGetSerializedData(ADR(out),SIZEOF(out));

AssertEquals(
	Expected := expected,
	Actual := out,
	Message := 'Did not produce the expected JSON string for the FileTime value'
);

TEST_FINISHED();
END_METHOD

METHOD PUBLIC TestAddKeyInt
VAR
	jsonSerializer : JsonSerializer;
	intValue : INT := 12345;
	out : STRING;
	expected : STRING := '{"data":12345}';
END_VAR
TEST('TestAddKeyInt');

jsonSerializer.StartObject();
jsonSerializer.AddKeyInt('data',intValue);
jsonSerializer.EndObject();

jsonSerializer.TryGetSerializedData(ADR(out),SIZEOF(out));

AssertEquals(
	Expected := expected,
	Actual := out,
	Message := 'Did not produce the expected JSON string for the INT value'
);

TEST_FINISHED();
END_METHOD

METHOD PUBLIC TestAddKeyLint
VAR
	jsonSerializer : JsonSerializer;
	lintValue : LINT := 9223372036854775807;
	out : STRING;
	expected : STRING := '{"data":9223372036854775807}';
END_VAR
TEST('TestAddKeyLint');

jsonSerializer.StartObject();
jsonSerializer.AddKeyLint('data',lintValue);
jsonSerializer.EndObject();

jsonSerializer.TryGetSerializedData(ADR(out),SIZEOF(out));

AssertEquals(
	Expected := expected,
	Actual := out,
	Message := 'Did not produce the expected JSON string for the LINT value'
);

TEST_FINISHED();
END_METHOD

METHOD PUBLIC TestAddKeyLreal
VAR
	jsonSerializer : JsonSerializer;
	lrealValue : LREAL := 123456.789;
	out : STRING;
	expected : STRING := '{"data":123456.789}';
END_VAR
TEST('TestAddKeyLreal');

jsonSerializer.StartObject();
jsonSerializer.AddKeyLreal('data',lrealValue);
jsonSerializer.EndObject();

jsonSerializer.TryGetSerializedData(ADR(out),SIZEOF(out));

AssertEquals(
	Expected := expected,
	Actual := out,
	Message := 'Did not produce the expected JSON string for the LREAL value'
);

TEST_FINISHED();
END_METHOD

METHOD PUBLIC TestAddKeyLreal_Max
VAR
	jsonSerializer : JsonSerializer;
	lrealValue : LREAL := DatatypeLimits.LREAL_MAX_VALUE;
	out : STRING;
	expected : STRING := '{"data":1.7976931348623157e308}';
END_VAR
TEST('TestAddKeyLreal_Max');

jsonSerializer.StartObject();
jsonSerializer.AddKeyLreal('data',lrealValue);
jsonSerializer.EndObject();

jsonSerializer.TryGetSerializedData(ADR(out),SIZEOF(out));

AssertEquals(
	Expected := expected,
	Actual := out,
	Message := 'Did not produce the expected JSON string for the LREAL value'
);

TEST_FINISHED();
END_METHOD

METHOD PUBLIC TestAddKeyLtime
VAR
	jsonSerializer : JsonSerializer;
	ltimeValue : LTIME := LTIME#100D2H30M40S500MS600US700NS;
	out : STRING;
	expected : STRING := '{"data":"LTIME#100d2h30m40s500ms600us700ns"}';
END_VAR
TEST('TestAddKeyLtime');

jsonSerializer.StartObject();
jsonSerializer.AddKeyLtime('data',ltimeValue);
jsonSerializer.EndObject();

jsonSerializer.TryGetSerializedData(ADR(out),SIZEOF(out));

AssertEquals(
	Expected := expected,
	Actual := out,
	Message := 'Did not produce the expected JSON string for the LTIME value'
);

TEST_FINISHED();
END_METHOD

METHOD PUBLIC TestAddKeyLword
VAR
	jsonSerializer : JsonSerializer;
	lwordValue : LWORD := 9223372036854775807;
	out : STRING;
	expected : STRING := '{"data":9223372036854775807}';
END_VAR
TEST('TestAddKeyLword');

jsonSerializer.StartObject();
jsonSerializer.AddKeyLword('data',lwordValue);
jsonSerializer.EndObject();

jsonSerializer.TryGetSerializedData(ADR(out),SIZEOF(out));

AssertEquals(
	Expected := expected,
	Actual := out,
	Message := 'Did not produce the expected JSON string for the LWORD value'
);

TEST_FINISHED();
END_METHOD

METHOD PUBLIC TestAddKeyNull
VAR
	jsonSerializer : JsonSerializer;
	out : STRING;
	expected : STRING := '{"data":null}';
END_VAR
TEST('TestAddKeyNull');

jsonSerializer.StartObject();
jsonSerializer.AddKeyNull('data');
jsonSerializer.EndObject();

jsonSerializer.TryGetSerializedData(ADR(out),SIZEOF(out));

AssertEquals(
	Expected := expected,
	Actual := out,
	Message := 'Did not produce the expected JSON string for the NULL value'
);

TEST_FINISHED();
END_METHOD

METHOD PUBLIC TestAddKeyObject
VAR
	jsonSerializer : JsonSerializer;
	user : MockSerializableUserObject(Name := 'alice', Age := 40);
	out : STRING;
	expected : STRING := '{"data":{"Name":"alice","Age":40}}';
END_VAR
TEST('TestAddKeyObject');

jsonSerializer.StartObject();
jsonSerializer.AddKeyObject('data',user);
jsonSerializer.EndObject();

jsonSerializer.TryGetSerializedData(ADR(out),SIZEOF(out));

AssertEquals(
	Expected := expected,
	Actual := out,
	Message := 'Did not produce the expected JSON string for the Object value'
);

TEST_FINISHED();
END_METHOD

METHOD PUBLIC TestAddKeyObject_Array
VAR
	jsonSerializer : JsonSerializer;
	user : MockSerializableArray(Name := 'alice', Age := 40);
	out : STRING;
	expected : STRING := '{"data":["alice",40]}';
END_VAR
TEST('TestAddKeyObject_Array');

jsonSerializer.StartObject();
jsonSerializer.AddKeyObject('data',user);
jsonSerializer.EndObject();

jsonSerializer.TryGetSerializedData(ADR(out),SIZEOF(out));

AssertEquals(
	Expected := expected,
	Actual := out,
	Message := 'Did not produce the expected JSON string for the Object value'
);

TEST_FINISHED();
END_METHOD

METHOD PUBLIC TestAddKeyRawJson
VAR
	jsonSerializer : JsonSerializer;
	rawObject : STRING := '{"foo":"bar"}';
	out : STRING;
	expected : STRING := '{"data":{"foo":"bar"}}';
END_VAR
TEST('TestAddKeyRawJson');

jsonSerializer.StartObject();
jsonSerializer.AddKeyRawJson('data',rawObject);
jsonSerializer.EndObject();

jsonSerializer.TryGetSerializedData(ADR(out),SIZEOF(out));

AssertEquals(
	Expected := expected,
	Actual := out,
	Message := 'Did not produce the expected JSON string for the raw object value'
);

TEST_FINISHED();
END_METHOD

METHOD PUBLIC TestAddKeyReal
VAR
	jsonSerializer : JsonSerializer;
	realValue : REAL := 123.4;
	out : STRING;
	expected : STRING := '{"data":123.4000015258789}'; // this has been adapted to support more decimal places, due to the issue with REAL conversion in TwinCAT 4024.56
END_VAR
TEST('TestAddKeyReal');

jsonSerializer.StartObject();
jsonSerializer.AddKeyReal('data',realValue);
jsonSerializer.EndObject();

jsonSerializer.TryGetSerializedData(ADR(out),SIZEOF(out));

AssertEquals(
	Expected := expected,
	Actual := out,
	Message := 'Did not produce the expected JSON string for the REAL value'
);

TEST_FINISHED();
END_METHOD

METHOD PUBLIC TestAddKeyReal_Max
VAR
	jsonSerializer : JsonSerializer;
	realValue : REAL := DatatypeLimits.REAL_MAX_VALUE;
	out : STRING;
	expected : STRING := '{"data":3.4028230607370967e38}'; // this has been adapted to support more decimal places, due to the issue with REAL conversion in TwinCAT 4024.56
END_VAR
TEST('TestAddKeyReal_Max');

jsonSerializer.StartObject();
jsonSerializer.AddKeyReal('data',realValue);
jsonSerializer.EndObject();

jsonSerializer.TryGetSerializedData(ADR(out),SIZEOF(out));

AssertEquals(
	Expected := expected,
	Actual := out,
	Message := 'Did not produce the expected JSON string for the REAL value'
);

TEST_FINISHED();
END_METHOD

METHOD PUBLIC TestAddKeySint
VAR
	jsonSerializer : JsonSerializer;
	sintValue : SINT := 123;
	out : STRING;
	expected : STRING := '{"data":123}';
END_VAR
TEST('TestAddKeySint');

jsonSerializer.StartObject();
jsonSerializer.AddKeySint('data',sintValue);
jsonSerializer.EndObject();

jsonSerializer.TryGetSerializedData(ADR(out),SIZEOF(out));

AssertEquals(
	Expected := expected,
	Actual := out,
	Message := 'Did not produce the expected JSON string for the SINT value'
);

TEST_FINISHED();
END_METHOD

METHOD PUBLIC TestAddKeyString
VAR
	jsonSerializer : JsonSerializer;
	stringValue : STRING := 'foobar';
	out : STRING;
	expected : STRING := '{"data":"foobar"}';
END_VAR
TEST('TestAddKeyString');

jsonSerializer.StartObject();
jsonSerializer.AddKeyString('data',stringValue);
jsonSerializer.EndObject();

jsonSerializer.TryGetSerializedData(ADR(out),SIZEOF(out));

AssertEquals(
	Expected := expected,
	Actual := out,
	Message := 'Did not produce the expected JSON string for the STRING value'
);

TEST_FINISHED();
END_METHOD

METHOD PUBLIC TestAddKeyStringByRef
VAR
	jsonSerializer : JsonSerializer;
	stringValue : T_MAXSTRING := '1234567890123456789012345678901234567890123456789012345678901234567890123456789012345678901234567890';
	out : T_MAXSTRING;
	expected : T_MAXSTRING := '{"data":"1234567890123456789012345678901234567890123456789012345678901234567890123456789012345678901234567890"}';
END_VAR
TEST('TestAddKeyStringByRef');

jsonSerializer.StartObject();
jsonSerializer.AddKeyStringByRef('data',stringValue);
jsonSerializer.EndObject();

jsonSerializer.TryGetSerializedData(ADR(out),SIZEOF(out));

AssertEquals(
	Expected := expected,
	Actual := out,
	Message := 'Did not produce the expected JSON string for the STRING using reference value'
);

TEST_FINISHED();
END_METHOD

METHOD PUBLIC TestAddKeyTime
VAR
	jsonSerializer : JsonSerializer;
	timeValue : TIME := T#49D17H2M47S295MS;
	out : STRING;
	expected : STRING := '{"data":"T#49d17h2m47s295ms"}';
END_VAR
TEST('TestAddKeyTime');

jsonSerializer.StartObject();
jsonSerializer.AddKeyTime('data',timeValue);
jsonSerializer.EndObject();

jsonSerializer.TryGetSerializedData(ADR(out),SIZEOF(out));

AssertEquals(
	Expected := expected,
	Actual := out,
	Message := 'Did not produce the expected JSON string for the TIME value'
);

TEST_FINISHED();
END_METHOD

METHOD PUBLIC TestAddKeyTod
VAR
	jsonSerializer : JsonSerializer;
	todValue : TOD := TOD#23:01:23.456;
	out : STRING;
	expected : STRING := '{"data":"TOD#23:01:23.456"}';
END_VAR
TEST('TestAddKeyTod');

jsonSerializer.StartObject();
jsonSerializer.AddKeyTod('data',todValue);
jsonSerializer.EndObject();

jsonSerializer.TryGetSerializedData(ADR(out),SIZEOF(out));

AssertEquals(
	Expected := expected,
	Actual := out,
	Message := 'Did not produce the expected JSON string for the TOD value'
);

TEST_FINISHED();
END_METHOD

METHOD PUBLIC TestAddKeyUdint
VAR
	jsonSerializer : JsonSerializer;
	udintValue : UDINT := 123456;
	out : STRING;
	expected : STRING := '{"data":123456}';
END_VAR
TEST('TestAddKeyUdint');

jsonSerializer.StartObject();
jsonSerializer.AddKeyUdint('data',udintValue);
jsonSerializer.EndObject();

jsonSerializer.TryGetSerializedData(ADR(out),SIZEOF(out));

AssertEquals(
	Expected := expected,
	Actual := out,
	Message := 'Did not produce the expected JSON string for the UDINT value'
);

TEST_FINISHED();
END_METHOD

METHOD PUBLIC TestAddKeyUint
VAR
	jsonSerializer : JsonSerializer;
	uintValue : UINT := 12345;
	out : STRING;
	expected : STRING := '{"data":12345}';
END_VAR
TEST('TestAddKeyUint');

jsonSerializer.StartObject();
jsonSerializer.AddKeyUint('data',uintValue);
jsonSerializer.EndObject();

jsonSerializer.TryGetSerializedData(ADR(out),SIZEOF(out));

AssertEquals(
	Expected := expected,
	Actual := out,
	Message := 'Did not produce the expected JSON string for the UINT value'
);

TEST_FINISHED();
END_METHOD

METHOD PUBLIC TestAddKeyUlint
VAR
	jsonSerializer : JsonSerializer;
	ulintValue : ULINT := 9223372036854775807;
	out : STRING;
	expected : STRING := '{"data":9223372036854775807}';
END_VAR
TEST('TestAddKeyUlint');

jsonSerializer.StartObject();
jsonSerializer.AddKeyUlint('data',ulintValue);
jsonSerializer.EndObject();

jsonSerializer.TryGetSerializedData(ADR(out),SIZEOF(out));

AssertEquals(
	Expected := expected,
	Actual := out,
	Message := 'Did not produce the expected JSON string for the ULINT value'
);

TEST_FINISHED();
END_METHOD

METHOD PUBLIC TestAddKeyUsint
VAR
	jsonSerializer : JsonSerializer;
	usintValue : USINT := 123;
	out : STRING;
	expected : STRING := '{"data":123}';
END_VAR
TEST('TestAddKeyUsint');

jsonSerializer.StartObject();
jsonSerializer.AddKeyUsint('data',usintValue);
jsonSerializer.EndObject();

jsonSerializer.TryGetSerializedData(ADR(out),SIZEOF(out));

AssertEquals(
	Expected := expected,
	Actual := out,
	Message := 'Did not produce the expected JSON string for the USINT value'
);

TEST_FINISHED();
END_METHOD

METHOD PUBLIC TestAddKeyWord
VAR
	jsonSerializer : JsonSerializer;
	wordValue : WORD := 12345;
	out : STRING;
	expected : STRING := '{"data":12345}';
END_VAR
TEST('TestAddKeyWord');

jsonSerializer.StartObject();
jsonSerializer.AddKeyWord('data',wordValue);
jsonSerializer.EndObject();

jsonSerializer.TryGetSerializedData(ADR(out),SIZEOF(out));

AssertEquals(
	Expected := expected,
	Actual := out,
	Message := 'Did not produce the expected JSON string for the WORD value'
);

TEST_FINISHED();
END_METHOD

METHOD PUBLIC TestAddLint
VAR
	jsonSerializer : JsonSerializer;
	lintValue : LINT := 9223372036854775807;
	out : STRING;
	expected : STRING := '9223372036854775807';
END_VAR
TEST('TestAddLint');

jsonSerializer.AddLint(lintValue);
jsonSerializer.TryGetSerializedData(ADR(out),SIZEOF(out));

AssertEquals(
	Expected := expected,
	Actual := out,
	Message := 'Did not produce the expected JSON string for the LINT value'
);

TEST_FINISHED();
END_METHOD

METHOD PUBLIC TestAddLreal
VAR
	jsonSerializer : JsonSerializer;
	lrealValue : LREAL := 123456.789;
	out : STRING;
	expected : STRING := '123456.789';
END_VAR
TEST('TestAddLReal');

jsonSerializer.AddLreal(lrealValue);
jsonSerializer.TryGetSerializedData(ADR(out),SIZEOF(out));

AssertEquals(
	Expected := expected,
	Actual := out,
	Message := 'Did not produce the expected JSON string for the LREAL value'
);

TEST_FINISHED();
END_METHOD

METHOD PUBLIC TestAddLtime
VAR
	jsonSerializer : JsonSerializer;
	ltimeValue : LTIME := LTIME#100D2H30M40S500MS600US700NS;
	out : STRING;
	expected : STRING := '"LTIME#100d2h30m40s500ms600us700ns"';
END_VAR
TEST('TestAddLtime');

jsonSerializer.AddLtime(ltimeValue);
jsonSerializer.TryGetSerializedData(ADR(out),SIZEOF(out));

AssertEquals(
	Expected := expected,
	Actual := out,
	Message := 'Did not produce the expected JSON string for the LTIME value'
);

TEST_FINISHED();
END_METHOD

METHOD PUBLIC TestAddLword
VAR
	jsonSerializer : JsonSerializer;
	lwordValue : LWORD := 9223372036854775807;
	out : STRING;
	expected : STRING := '9223372036854775807';
END_VAR
TEST('TestAddLword');

jsonSerializer.AddLword(lwordValue);
jsonSerializer.TryGetSerializedData(ADR(out),SIZEOF(out));

AssertEquals(
	Expected := expected,
	Actual := out,
	Message := 'Did not produce the expected JSON string for the LWORD value'
);

TEST_FINISHED();
END_METHOD

METHOD PUBLIC TestAddNull
VAR
	jsonSerializer : JsonSerializer;
	out : STRING;
	expected : STRING := 'null';
END_VAR
TEST('TestAddNull');

jsonSerializer.AddNull();
jsonSerializer.TryGetSerializedData(ADR(out),SIZEOF(out));

AssertEquals(
	Expected := expected,
	Actual := out,
	Message := 'Did not produce the expected JSON string for the NULL value'
);

TEST_FINISHED();
END_METHOD

METHOD PUBLIC TestAddObject
VAR
	jsonSerializer : JsonSerializer;
	user : MockSerializableUserObject(Name := 'alice', Age := 40);
	out : STRING;
	expected : STRING := '{"Name":"alice","Age":40}';
END_VAR
TEST('TestAddObject');

jsonSerializer.AddObject(user);
jsonSerializer.TryGetSerializedData(ADR(out),SIZEOF(out));

AssertEquals(
	Expected := expected,
	Actual := out,
	Message := 'Did not produce the expected JSON string for the Object value'
);

TEST_FINISHED();
END_METHOD

METHOD PUBLIC TestAddObjects
VAR
	jsonSerializer : JsonSerializer;
	user1 : MockSerializableUserObject(Name := 'alice', Age := 40);
    user2 : MockSerializableUserObject(Name := 'bob', Age := 50);
	out : STRING;
	expected : STRING := '{"users":[{"Name":"alice","Age":40},{"Name":"bob","Age":50}]}';
END_VAR
TEST('TestAddObjects');

jsonSerializer.StartObject();
jsonSerializer.AddKey('users');
jsonSerializer.StartArray();
jsonSerializer.AddObject(user1);
jsonSerializer.AddObject(user2);
jsonSerializer.EndArray();
jsonSerializer.EndObject();
jsonSerializer.TryGetSerializedData(ADR(out),SIZEOF(out));

AssertEquals(
	Expected := expected,
	Actual := out,
	Message := 'Did not produce the expected JSON string for the Object value'
);

TEST_FINISHED();
END_METHOD

METHOD PUBLIC TestAddRawJson
VAR
	jsonSerializer : JsonSerializer;
	rawObject : STRING := '{"foo":"bar"}';
	out : STRING;
	expected : STRING := '{"foo":"bar"}';
END_VAR
TEST('TestAddRawJson');

jsonSerializer.AddRawJson(rawObject);
jsonSerializer.TryGetSerializedData(ADR(out),SIZEOF(out));

AssertEquals(
	Expected := expected,
	Actual := out,
	Message := 'Did not produce the expected JSON string for the raw object value'
);

TEST_FINISHED();
END_METHOD

METHOD PUBLIC TestAddReal
VAR
	jsonSerializer : JsonSerializer;
	realValue : REAL := 123.4;
	out : STRING;
	expected : STRING := '123.4000015258789'; // this has been adapted to support more decimal places, due to the issue with REAL conversion in TwinCAT 4024.56
END_VAR
TEST('TestAddReal');

jsonSerializer.AddReal(realValue);
jsonSerializer.TryGetSerializedData(ADR(out),SIZEOF(out));

AssertEquals(
	Expected := expected,
	Actual := out,
	Message := 'Did not produce the expected JSON string for the REAL value'
);

TEST_FINISHED();
END_METHOD

METHOD PUBLIC TestAddSint
VAR
	jsonSerializer : JsonSerializer;
	intValue : SINT := 123;
	out : STRING;
	expected : STRING := '123';
END_VAR
TEST('TestAddSint');

jsonSerializer.AddSint(intValue);
jsonSerializer.TryGetSerializedData(ADR(out),SIZEOF(out));

AssertEquals(
	Expected := expected,
	Actual := out,
	Message := 'Did not produce the expected JSON string for the SINT value'
);

TEST_FINISHED();
END_METHOD

METHOD PUBLIC TestAddString
VAR
	jsonSerializer : JsonSerializer;
	stringValue : STRING := 'foobar';
	out : STRING;
	expected : STRING := '"foobar"';
END_VAR
TEST('TestAddString');

jsonSerializer.AddString(stringValue);
jsonSerializer.TryGetSerializedData(ADR(out),SIZEOF(out));

AssertEquals(
	Expected := expected,
	Actual := out,
	Message := 'Did not produce the expected JSON string for the STRING value'
);

TEST_FINISHED();
END_METHOD

METHOD PUBLIC TestAddStringByRef
VAR
	jsonSerializer : JsonSerializer;
	stringValue : T_MAXSTRING := '1234567890123456789012345678901234567890123456789012345678901234567890123456789012345678901234567890';
	out : T_MAXSTRING;
	expected : T_MAXSTRING := '"1234567890123456789012345678901234567890123456789012345678901234567890123456789012345678901234567890"';
END_VAR
TEST('TestAddStringByRef');

jsonSerializer.AddStringByRef(stringValue);
jsonSerializer.TryGetSerializedData(ADR(out),SIZEOF(out));

AssertEquals(
	Expected := expected,
	Actual := out,
	Message := 'Did not produce the expected JSON string for the STRING using reference value'
);

TEST_FINISHED();
END_METHOD

METHOD PUBLIC TestAddTime
VAR
	jsonSerializer : JsonSerializer;
	timeValue : TIME := T#49D17H2M47S295MS;
	out : STRING;
	expected : STRING := '"T#49d17h2m47s295ms"';
END_VAR
TEST('TestAddTime');

jsonSerializer.AddTime(timeValue);
jsonSerializer.TryGetSerializedData(ADR(out),SIZEOF(out));

AssertEquals(
	Expected := expected,
	Actual := out,
	Message := 'Did not produce the expected JSON string for the TIME value'
);

TEST_FINISHED();
END_METHOD

METHOD PUBLIC TestAddTod
VAR
	jsonSerializer : JsonSerializer;
	todValue : TOD := TOD#23:01:23.456;
	out : STRING;
	expected : STRING := '"TOD#23:01:23.456"';
END_VAR
TEST('TestAddTod');

jsonSerializer.AddTod(todValue);
jsonSerializer.TryGetSerializedData(ADR(out),SIZEOF(out));

AssertEquals(
	Expected := expected,
	Actual := out,
	Message := 'Did not produce the expected JSON string for the TOD value'
);

TEST_FINISHED();
END_METHOD

METHOD PUBLIC TestAddUdint
VAR
	jsonSerializer : JsonSerializer;
	udintValue : UDINT := 123456;
	out : STRING;
	expected : STRING := '123456';
END_VAR
TEST('TestAddUdint');

jsonSerializer.AddUdint(udintValue);
jsonSerializer.TryGetSerializedData(ADR(out),SIZEOF(out));

AssertEquals(
	Expected := expected,
	Actual := out,
	Message := 'Did not produce the expected JSON string for the UDINT value'
);

TEST_FINISHED();
END_METHOD

METHOD PUBLIC TestAddUint
VAR
	jsonSerializer : JsonSerializer;
	uintValue : UINT := 12345;
	out : STRING;
	expected : STRING := '12345';
END_VAR
TEST('TestAddUint');


jsonSerializer.AddUint(uintValue);
jsonSerializer.TryGetSerializedData(ADR(out),SIZEOF(out));

AssertEquals(
	Expected := expected,
	Actual := out,
	Message := 'Did not produce the expected JSON string for the UINT value'
);

TEST_FINISHED();
END_METHOD

METHOD PUBLIC TestAddUlint
VAR
	jsonSerializer : JsonSerializer;
	ulintValue : ULINT := 9223372036854775807;
	out : STRING;
	expected : STRING := '9223372036854775807';
END_VAR
TEST('TestAddUlint');

jsonSerializer.AddUlint(ulintValue);
jsonSerializer.TryGetSerializedData(ADR(out),SIZEOF(out));

AssertEquals(
	Expected := expected,
	Actual := out,
	Message := 'Did not produce the expected JSON string for the ULINT value'
);

TEST_FINISHED();
END_METHOD

METHOD PUBLIC TestAddUsint
VAR
	jsonSerializer : JsonSerializer;
	usintValue : USINT := 123;
	out : STRING;
	expected : STRING := '123';
END_VAR
TEST('TestAddUsint');

jsonSerializer.AddUsint(usintValue);
jsonSerializer.TryGetSerializedData(ADR(out),SIZEOF(out));

AssertEquals(
	Expected := expected,
	Actual := out,
	Message := 'Did not produce the expected JSON string for the USINT value'
);

TEST_FINISHED();
END_METHOD

METHOD PUBLIC TestAddWord
VAR
	jsonSerializer : JsonSerializer;
	wordValue : WORD := 12345;
	out : STRING;
	expected : STRING := '12345';
END_VAR
TEST('TestAddWord');

jsonSerializer.AddWord(wordValue);
jsonSerializer.TryGetSerializedData(ADR(out),SIZEOF(out));

AssertEquals(
	Expected := expected,
	Actual := out,
	Message := 'Did not produce the expected JSON string for the WORD value'
);

TEST_FINISHED();
END_METHOD

METHOD PUBLIC TestClone
VAR
	jsonSerializer : JsonSerializer;
	clone : I_Serializer;
	rawObject : STRING := '{"foo":"bar"}';
	out : STRING;
	expected : STRING := '{"foo":"bar"}';
END_VAR
TEST('TestClone');

// add something to the original 
jsonSerializer.AddRawJson(rawObject);

// deep clone
clone := jsonSerializer.Clone();

// reset the original
jsonSerializer.Reset();

// retreive the data from the clone
clone.TryGetSerializedData(ADR(out),SIZEOF(out));

// clones are __NEW so must be disposed
clone.Dispose();

AssertEquals(
	Expected := expected,
	Actual := out,
	Message := 'Did not create a deep copy clone'
);

TEST_FINISHED();
END_METHOD

METHOD PUBLIC TestGetSerializedDataLengthEmpty
VAR
	jsonSerializer : JsonSerializer;
	rawObject : STRING := '';
	length : UDINT;
	expected : UDINT := 0;
END_VAR
TEST('TestGetSerializedDataLengthEmpty');

length := jsonSerializer.GetSerializedDataLength();

AssertEquals(
	Expected := expected,
	Actual := length,
	Message := 'Did not produce the expected JSON string length'
);

TEST_FINISHED();
END_METHOD

METHOD PUBLIC TestGetSerializedDataLengthWithEmptyObject
VAR
	jsonSerializer : JsonSerializer;
	rawObject : STRING := '{}';
	length : UDINT;
	expected : UDINT := 3;
END_VAR
TEST('TestGetSerializedDataLengthWithEmptyObject');

jsonSerializer.AddRawJson(rawObject);
length := jsonSerializer.GetSerializedDataLength();

AssertEquals(
	Expected := expected,
	Actual := length,
	Message := 'Did not produce the expected JSON string length'
);

TEST_FINISHED();
END_METHOD

METHOD PUBLIC TestGetSerializedDataLengthWithSimpleObject
VAR
	jsonSerializer : JsonSerializer;
	rawObject : STRING := '{"foo":"bar"}';
	length : UDINT;
	expected : UDINT := 14;
END_VAR
TEST('TestGetSerializedDataLength');

jsonSerializer.AddRawJson(rawObject);
length := jsonSerializer.GetSerializedDataLength();

AssertEquals(
	Expected := expected,
	Actual := length,
	Message := 'Did not produce the expected JSON string length'
);

TEST_FINISHED();
END_METHOD

METHOD PUBLIC TestReset
VAR
	jsonSerializer : JsonSerializer;
	rawObject : STRING := '{"foo":"bar"}';
	out : STRING;
	expected : STRING := '';
END_VAR
TEST('TestReset');

jsonSerializer.AddRawJson(rawObject);
jsonSerializer.Reset();
jsonSerializer.TryGetSerializedData(ADR(out),SIZEOF(out));

AssertEquals(
	Expected := expected,
	Actual := out,
	Message := 'Did not reset'
);

TEST_FINISHED();
END_METHOD

METHOD PUBLIC TestSerializeArray
VAR
	jsonSerializer : JsonSerializer;
	out : STRING;
	expected : STRING := '[123,true,"foobar",null]';
END_VAR
TEST('TestSerializeArray');

jsonSerializer.StartArray();
jsonSerializer.AddDint(123);
jsonSerializer.AddBool(TRUE);
jsonSerializer.AddString('foobar');
jsonSerializer.AddNull();
jsonSerializer.EndArray();

jsonSerializer.TryGetSerializedData(ADR(out),SIZEOF(out));

AssertEquals(
	Expected := expected,
	Actual := out,
	Message := 'Did not produce the expected JSON string for the array'
);

TEST_FINISHED();
END_METHOD

METHOD PUBLIC TestSerializeObject
VAR
	jsonSerializer : JsonSerializer;
	out : STRING;
	expected : STRING := '{"dint":123,"bool":true,"string":"foobar","null":null}';
END_VAR
TEST('TestSerializeObject');

jsonSerializer.StartObject();
jsonSerializer.AddKeyDint('dint',123);
jsonSerializer.AddKeyBool('bool',TRUE);
jsonSerializer.AddKeyString('string','foobar');
jsonSerializer.AddKeyNull('null');
jsonSerializer.EndObject();

jsonSerializer.TryGetSerializedData(ADR(out),SIZEOF(out));

AssertEquals(
	Expected := expected,
	Actual := out,
	Message := 'Did not produce the expected JSON string for the object'
);

TEST_FINISHED();
END_METHOD

END_FUNCTION_BLOCK

// ---- Tests/Mocks/MockSerializableUserObject.TcPOU
FUNCTION_BLOCK MockSerializableUserObject IMPLEMENTS I_Serializable
VAR
	_name : STRING;
	_age : INT;
END_VAR

PROPERTY PUBLIC Age : INT
GET
Age := _age;
END_GET
SET
_age := Age;
END_SET
END_PROPERTY

METHOD FB_init : BOOL
VAR_INPUT
	bInitRetains : BOOL; // if TRUE, the retain variables are initialized (warm start / cold start)
	bInCopyCode : BOOL;  // if TRUE, the instance afterwards gets moved into the copy code (online change)
	Name : STRING;
	Age : INT;
END_VAR
_name := Name;
_age := Age;
END_METHOD

PROPERTY PUBLIC Name : STRING
GET
Name := _name;
END_GET
SET
_name := Name;
END_SET
END_PROPERTY

METHOD SerializeWith
VAR_INPUT
	Serializer : I_Serializer;
END_VAR
Serializer.StartObject().AddKeyString('Name',_name).AddKeyInt('Age',_age).EndObject();
END_METHOD

END_FUNCTION_BLOCK

// ---- Tests/Mocks/MockSerializableArray.TcPOU
FUNCTION_BLOCK MockSerializableArray IMPLEMENTS I_Serializable
VAR
	_name : STRING;
	_age : INT;
END_VAR

PROPERTY PUBLIC Age : INT
GET
Age := _age;
END_GET
SET
_age := Age;
END_SET
END_PROPERTY

METHOD FB_init : BOOL
VAR_INPUT
	bInitRetains : BOOL; // if TRUE, the retain variables are initialized (warm start / cold start)
	bInCopyCode : BOOL;  // if TRUE, the instance afterwards gets moved into the copy code (online change)
	Name : STRING;
	Age : INT;
END_VAR
_name := Name;
_age := Age;
END_METHOD

PROPERTY PUBLIC Name : STRING
GET
Name := _name;
END_GET
SET
_name := Name;
END_SET
END_PROPERTY

METHOD SerializeWith
VAR_INPUT
	Serializer : I_Serializer;
END_VAR
Serializer.StartArray().AddString(_name).AddInt(_age).EndArray();
END_METHOD

END_FUNCTION_BLOCK

// ---- Tests/JsonDeserializer_TestSuite.TcPOU
FUNCTION_BLOCK JsonDeserializer_TestSuite EXTENDS TcUnit.FB_TestSuite

TestClone();
TestReset();
TestGetArray();
TestGetKeyArray();
TestGetKeyObject();
TestGetObject();
TestTryGetBase64();
TestTryGetBoolWithFalseValue();
TestTryGetBoolWithTrueValue();
TestTryGetByte();
TestTryGetHexAsBytes();
TestTryGetDateTime();
TestTryGetDcTime();
TestTryGetDint();
TestTryGetDword();
TestTryGetFileTime();
TestTryGetInt();
TestTryGetKeyBase64();
TestTryGetKeyBoolWithFalseBoolVariable();
TestTryGetKeyBoolWithTrueBoolVariable();
TestTryGetKeyByte();
TestTryGetKeyHexAsBytes();
TestTryGetKeyDateTime();
TestTryGetKeyDcTime();
TestTryGetKeyDint();
TestTryGetKeyDword();
TestTryGetKeyFileTime();
TestTryGetKeyInt();
TestTryGetKeyLint();
TestTryGetKeyLreal();
TestTryGetKeyLtime();
TestTryGetKeyLword();
TestTryDeserializeKeyToObject();
TestTryDeserializeKeyToObjectFailsWithMissingKey();
TestTryDeserializeKeyToObjectFailsWithInvalidKey();
TestTryGetKeyReal();
TestTryGetKeySint();
TestTryGetKeyString();
TestTryGetKeyTime();
TestTryGetKeyTod();
TestTryGetKeyUdint();
TestTryGetKeyUint();
TestTryGetKeyUlint();
TestTryGetKeyUsint();
TestTryGetKeyWord();
TestTryGetLint();
TestTryGetLreal();
TestTryGetLtime();
TestTryGetLword();
TestTryDeserializeToObject();
TestTryGetReal();
TestTryGetSint();
TestTryGetString();
TestTryGetTime();
TestTryGetTod();
TestTryGetUdint();
TestTryGetUint();
TestTryGetUlint();
TestTryGetUsint();
TestTryGetWord();

METHOD PUBLIC TestClone
VAR
	jsonDeserializer : JsonDeserializer;
	clone : I_Deserializer;
    json : STRING := '{"data":100}';
    out : BYTE;
	feedback : DeserializerFeedback;
	hasDeserializer : BOOL;
    expected : BYTE := 100;
END_VAR
TEST('TestClone');

// add something to the original 
jsonDeserializer.TryLoad(json);

// deep clone
clone := jsonDeserializer.Clone();

// reset the original
jsonDeserializer.Reset();

// retreive the data from the clone
clone.TryGetKeyByte('data', out, feedback);

// clones are __NEW so must be disposed
clone.Dispose();

AssertEquals(
	Expected := expected,
	Actual := out,
	Message := 'Did not create a deep copy clone'
);

TEST_FINISHED();
END_METHOD

METHOD PUBLIC TestGetArray
VAR
    jsonDeserializer : JsonDeserializer;
	arrayDeserializer : I_Deserializer;
	elementDeserializer : I_Deserializer;
    json : STRING := '[100,200,300]';
    out : BYTE;
	feedback : DeserializerFeedback;
	hasArrayDeserializer : BOOL;
	hasElementDeserializer : BOOL;
    expected : BYTE := 100;
END_VAR
TEST('TestGetArray');

jsonDeserializer.TryLoad(json);
arrayDeserializer := jsonDeserializer.GetArray();

hasArrayDeserializer := arrayDeserializer <> 0;

IF hasArrayDeserializer THEN
	elementDeserializer := arrayDeserializer.GetElementByIndex(0);
END_IF

AssertTrue(
	Condition := hasArrayDeserializer,
	Message := 'Did not return deserializer for array'
);

hasElementDeserializer := elementDeserializer <> 0;

IF hasElementDeserializer THEN
	elementDeserializer.TryGetByte(out, feedback);
END_IF

AssertTrue(
	Condition := hasElementDeserializer,
	Message := 'Did not return deserializer for element'
);

AssertEquals(
    Expected := expected,
    Actual := out,
    Message := 'Did not produce the expected BYTE value from JSON array'
);

TEST_FINISHED();
END_METHOD

METHOD PUBLIC TestGetKeyArray
VAR
    jsonDeserializer : JsonDeserializer;
	arrayDeserializer : I_Deserializer;
	elementDeserializer : I_Deserializer;
    json : STRING := '{"myArray":[100,200,300]}';
    out : BYTE;
	feedback : DeserializerFeedback;
	hasArrayDeserializer : BOOL;
	hasElementDeserializer : BOOL;
    expected : BYTE := 100;
END_VAR
TEST('TestGetKeyArray');

jsonDeserializer.TryLoad(json);
arrayDeserializer := jsonDeserializer.GetKeyArray('myArray');

hasArrayDeserializer := arrayDeserializer <> 0;

IF hasArrayDeserializer THEN
	elementDeserializer := arrayDeserializer.GetElementByIndex(0);
END_IF

AssertTrue(
	Condition := hasArrayDeserializer,
	Message := 'Did not return deserializer for array'
);

hasElementDeserializer := elementDeserializer <> 0;

IF hasElementDeserializer THEN
	elementDeserializer.TryGetByte(out, feedback);
END_IF

AssertTrue(
	Condition := hasElementDeserializer,
	Message := 'Did not return deserializer for element'
);

AssertEquals(
    Expected := expected,
    Actual := out,
    Message := 'Did not produce the expected BYTE value from JSON array'
);

TEST_FINISHED();
END_METHOD

METHOD PUBLIC TestGetKeyObject
VAR
    jsonDeserializer : JsonDeserializer;
	objectDeserializer : I_Deserializer;
    json : STRING := '{"data":100}';
    out : BYTE;
	feedback : DeserializerFeedback;
	hasObjectDeserializer : BOOL;
    expected : BYTE := 100;
END_VAR
TEST('TestGetKeyObject');

jsonDeserializer.TryLoad(json);
objectDeserializer := jsonDeserializer.GetKeyObject('data');

hasObjectDeserializer := objectDeserializer <> 0;

IF hasObjectDeserializer THEN
	objectDeserializer.TryGetByte(out, feedback);
END_IF

AssertTrue(
	Condition := hasObjectDeserializer,
	Message := 'Did not return deserializer for object'
);

AssertEquals(
    Expected := expected,
    Actual := out,
    Message := 'Did not produce the expected BYTE value from JSON'
);

TEST_FINISHED();
END_METHOD

METHOD PUBLIC TestGetObject
VAR
    jsonDeserializer : JsonDeserializer;
	objectDeserializer : I_Deserializer;
    json : STRING := '{"data":100}';
    out : BYTE;
	feedback : DeserializerFeedback;
	hasObjectDeserializer : BOOL;
    expected : BYTE := 100;
END_VAR
TEST('TestGetObject');

jsonDeserializer.TryLoad(json);
objectDeserializer := jsonDeserializer.GetObject();

hasObjectDeserializer := objectDeserializer <> 0;

IF hasObjectDeserializer THEN
	objectDeserializer.TryGetKeyByte('data',out, feedback);
END_IF

AssertTrue(
	Condition := hasObjectDeserializer,
	Message := 'Did not return deserializer for object'
);

AssertEquals(
    Expected := expected,
    Actual := out,
    Message := 'Did not produce the expected BYTE value from JSON'
);

TEST_FINISHED();
END_METHOD

METHOD PUBLIC TestReset
VAR
	jsonDeserializer : JsonDeserializer;
    json : STRING := '100';
    out : BYTE;
	feedback : DeserializerFeedback;
    expected : BYTE := 0; 
END_VAR
TEST('TestReset');

jsonDeserializer.TryLoad(json);
jsonDeserializer.Reset();
jsonDeserializer.TryGetByte(out, feedback);

AssertEquals(
	Expected := expected,
	Actual := out,
	Message := 'Did not reset'
);

TEST_FINISHED();
END_METHOD

METHOD PUBLIC TestTryDeserializeKeyToObject
VAR
    jsonDeserializer : JsonDeserializer;
    json : STRING := '{"data":{"Name":"alice","Age":40}}';
    out : MockDeserializableUserObject;
	feedback : DeserializerFeedback;
    expectedName : STRING := 'alice';
	expectedAge : INT := 40;
	actualName : STRING;
	actualAge : INT;
END_VAR
TEST('TestTryDeserializeKeyToObject');
jsonDeserializer.TryLoad(json);
jsonDeserializer.TryDeserializeKeyToObject('data', out, feedback);

actualName := out.Name;
actualAge := out.Age;

AssertEquals(
    Expected := expectedName,
    Actual := actualName,
    Message := 'Did not produce the expected Object values from JSON'
);

AssertEquals(
    Expected := expectedAge,
    Actual := actualAge,
    Message := 'Did not produce the expected Object values from JSON'
);

TEST_FINISHED();
END_METHOD

METHOD PUBLIC TestTryDeserializeKeyToObjectFailsWithInvalidKey
VAR
    jsonDeserializer : JsonDeserializer;
    json : STRING := '{"data":{"Name":"alice","Age":40}}';
    out : MockDeserializableUserObject;
	feedback : DeserializerFeedback;
	result : BOOL;
END_VAR
TEST('TestTryDeserializeKeyToObjectFailsWithInvalidKey');
jsonDeserializer.TryLoad(json);
result := jsonDeserializer.TryDeserializeKeyToObject('', out, feedback);

AssertFalse(
	Condition := result,
	Message := 'Try returned true, even though key was invalid present');

TEST_FINISHED();
END_METHOD

METHOD PUBLIC TestTryDeserializeKeyToObjectFailsWithMissingKey
VAR
    jsonDeserializer : JsonDeserializer;
    json : STRING := '{"data":{"Name":"alice","Age":40}}';
    out : MockDeserializableUserObject;
	feedback : DeserializerFeedback;
	result : BOOL;
END_VAR
TEST('TestTryDeserializeKeyToObjectFailsWithMissingKey');
jsonDeserializer.TryLoad(json);
result := jsonDeserializer.TryDeserializeKeyToObject('test', out, feedback);

AssertFalse(
	Condition := result,
	Message := 'Try returned true, even though key was not present');

TEST_FINISHED();
END_METHOD

METHOD PUBLIC TestTryDeserializeToObject
VAR
    jsonDeserializer : JsonDeserializer;
    json : STRING := '{"Name":"alice","Age":40}';
    out : MockDeserializableUserObject;
	feedback : DeserializerFeedback;
    expectedName : STRING := 'alice';
	expectedAge : INT := 40;
	actualName : STRING;
	actualAge : INT;
END_VAR
TEST('TestTryDeserializeToObject');

jsonDeserializer.TryLoad(json);
jsonDeserializer.TryDeserializeToObject(out, feedback);

actualName := out.Name;
actualAge := out.Age;

AssertEquals(
    Expected := expectedName,
    Actual := actualName,
    Message := 'Did not produce the expected Object values from JSON'
);

AssertEquals(
    Expected := expectedAge,
    Actual := actualAge,
    Message := 'Did not produce the expected Object values from JSON'
);

TEST_FINISHED();
END_METHOD

METHOD PUBLIC TestTryGetBase64
VAR
	jsonDeserializer : JsonDeserializer;
	json : STRING := '"aGVsbG8="';
	out : ARRAY[0..4] OF BYTE;
	feedback : DeserializerFeedback;
	expected : ARRAY[0..4] OF BYTE := [104, 101, 108, 108, 111]; 
END_VAR
TEST('TestTryGetBase64');

jsonDeserializer.TryLoad(json);
jsonDeserializer.TryGetBase64(ADR(out), SIZEOF(out), feedback);

AssertEquals(
	Expected := expected,
	Actual := out,
	Message := 'Did not produce the expected Base64 encoded "hello" from JSON'
);

TEST_FINISHED();
END_METHOD

METHOD PUBLIC TestTryGetBoolWithFalseValue
VAR
	jsonDeserializer : JsonDeserializer;
	json : STRING := 'false';
	out : BOOL;
	feedback : DeserializerFeedback;
	expected : BOOL := FALSE;
END_VAR
TEST('TestTryGetBoolWithFalseValue');

jsonDeserializer.TryLoad(json);
jsonDeserializer.TryGetBool(out, feedback);

AssertEquals(
	Expected := expected,
	Actual := out,
	Message := 'Did not produce the expected JSON string for a false value'
);

TEST_FINISHED();
END_METHOD

METHOD PUBLIC TestTryGetBoolWithTrueValue
VAR
    jsonDeserializer : JsonDeserializer;
    json : STRING := 'true';
    out : BOOL;
	feedback : DeserializerFeedback;
    expected : BOOL := TRUE; 
END_VAR
TEST('TestTryGetBoolWithTrueValue');

jsonDeserializer.TryLoad(json);
jsonDeserializer.TryGetBool(out, feedback);

AssertEquals(
    Expected := expected,
    Actual := out,
    Message := 'Did not produce the expected true value from JSON'
);

TEST_FINISHED();
END_METHOD

METHOD PUBLIC TestTryGetByte
VAR
    jsonDeserializer : JsonDeserializer;
    json : STRING := '100';
    out : BYTE;
	feedback : DeserializerFeedback;
    expected : BYTE := 100; 
END_VAR
TEST('TestTryGetByte');

jsonDeserializer.TryLoad(json);
jsonDeserializer.TryGetByte(out, feedback);

AssertEquals(
    Expected := expected,
    Actual := out,
    Message := 'Did not produce the expected BYTE value from JSON'
);

TEST_FINISHED();
END_METHOD

METHOD PUBLIC TestTryGetDateTime
VAR
    jsonDeserializer : JsonDeserializer;
    json : STRING := '"2023-12-30T15:20:00"';
    out : DATE_AND_TIME;
	feedback : DeserializerFeedback;
    expected : DATE_AND_TIME := DT#2023-12-30-15:20:00; 
END_VAR
TEST('TestTryGetDateTime');

jsonDeserializer.TryLoad(json);
jsonDeserializer.TryGetDateTime(out, feedback);

AssertEquals(
    Expected := expected,
    Actual := out,
    Message := 'Did not produce the expected DATE_AND_TIME value from JSON'
);

TEST_FINISHED();
END_METHOD

METHOD PUBLIC TestTryGetDcTime
VAR
    jsonDeserializer : JsonDeserializer;
    json : STRING := '"2000-01-01T00:00:00.012345678"';
    out : DCTIME;
	feedback : DeserializerFeedback;
    expected : DCTIME := 12345678;
END_VAR
TEST('TestTryGetDcTime');

jsonDeserializer.TryLoad(json);
jsonDeserializer.TryGetDcTime(out, feedback);

AssertEquals(
    Expected := expected,
    Actual := out,
    Message := 'Did not produce the expected DCTIME value from JSON string'
);

TEST_FINISHED();
END_METHOD

METHOD PUBLIC TestTryGetDint
VAR
    jsonDeserializer : JsonDeserializer;
    json : STRING := '12345';
    out : DINT;
	feedback : DeserializerFeedback;
    expected : DINT := 12345;
END_VAR
TEST('TestTryGetDint');

jsonDeserializer.TryLoad(json);
jsonDeserializer.TryGetDint(out, feedback);

AssertEquals(
    Expected := expected,
    Actual := out,
    Message := 'Did not produce the expected DINT value from JSON'
);

TEST_FINISHED();
END_METHOD

METHOD PUBLIC TestTryGetDword
VAR
    jsonDeserializer : JsonDeserializer;
    json : STRING := '12345';
    out : DWORD;
	feedback : DeserializerFeedback;
    expected : DWORD := 12345;
END_VAR
TEST('TestTryGetDword');

jsonDeserializer.TryLoad(json);
jsonDeserializer.TryGetDword(out, feedback);

AssertEquals(
    Expected := expected,
    Actual := out,
    Message := 'Did not produce the expected DWORD value from JSON'
);

TEST_FINISHED();
END_METHOD

METHOD PUBLIC TestTryGetFileTime
VAR
    jsonDeserializer : JsonDeserializer;
    json : STRING := '"1601-01-01T00:00:01.2345678"';
    out : FILETIME;
	feedback : DeserializerFeedback;
    expected : FILETIME := 12345678; 
END_VAR
TEST('TestTryGetFileTime');

jsonDeserializer.TryLoad(json);
jsonDeserializer.TryGetFileTime(out, feedback);

AssertEquals(
    Expected := expected,
    Actual := out,
    Message := 'Did not produce the expected FILETIME value from JSON'
);

TEST_FINISHED();
END_METHOD

METHOD PUBLIC TestTryGetHexAsBytes
VAR
    jsonDeserializer : JsonDeserializer;
    json : STRING := '"baadf00d"';
    out : ARRAY[0..3] OF BYTE;
	feedback : DeserializerFeedback;
    expected : ARRAY[0..3] OF BYTE := [16#BA, 16#AD, 16#F0, 16#0D];
END_VAR
TEST('TestTryGetHexAsBytes');

jsonDeserializer.TryLoad(json);
jsonDeserializer.TryGetHexAsBytes(ADR(out), SIZEOF(out), feedback);

AssertEquals(
    Expected := expected,
    Actual := out,
    Message := 'Did not produce the expected binary data from JSON hexadecimal string'
);

TEST_FINISHED();
END_METHOD

METHOD PUBLIC TestTryGetInt
VAR
    jsonDeserializer : JsonDeserializer;
    json : STRING := '12345';
    out : INT;
	feedback : DeserializerFeedback;
    expected : INT := 12345;
END_VAR
TEST('TestTryGetInt');

jsonDeserializer.TryLoad(json);
jsonDeserializer.TryGetInt(out, feedback);

AssertEquals(
    Expected := expected,
    Actual := out,
    Message := 'Did not produce the expected INT value from JSON'
);

TEST_FINISHED();
END_METHOD

METHOD PUBLIC TestTryGetKeyBase64
VAR
    jsonDeserializer : JsonDeserializer;
    json : STRING := '{"data":"aGVsbG8="}';
    out : ARRAY[0..4] OF BYTE;
	feedback : DeserializerFeedback;
    expected : ARRAY[0..4] OF BYTE := [104, 101, 108, 108, 111];
END_VAR
TEST('TestTryGetKeyBase64');

jsonDeserializer.TryLoad(json);
jsonDeserializer.TryGetKeyBase64('data', ADR(out), SIZEOF(out), feedback);

AssertEquals(
    Expected := expected,
    Actual := out,
    Message := 'Did not produce the expected binary data from JSON Base64 encoded "hello"'
);

TEST_FINISHED();
END_METHOD

METHOD PUBLIC TestTryGetKeyBoolWithFalseBoolVariable
VAR
    jsonDeserializer : JsonDeserializer;
    json : STRING := '{"data":false}';
    out : BOOL;
	feedback : DeserializerFeedback;
    expected : BOOL := FALSE;
END_VAR
TEST('TestTryGetKeyBoolWithFalseBoolVariable');

jsonDeserializer.TryLoad(json);
jsonDeserializer.TryGetKeyBool('data', out, feedback);

AssertEquals(
    Expected := expected,
    Actual := out,
    Message := 'Did not produce the expected boolean value from JSON for a false value'
);

TEST_FINISHED();
END_METHOD

METHOD PUBLIC TestTryGetKeyBoolWithTrueBoolVariable
VAR
    jsonDeserializer : JsonDeserializer;
    json : STRING := '{"data":true}';
    out : BOOL;
	feedback : DeserializerFeedback;
    expected : BOOL := TRUE;
END_VAR
TEST('TestTryGetKeyBoolWithTrueBoolVariable');

jsonDeserializer.TryLoad(json);
jsonDeserializer.TryGetKeyBool('data', out, feedback);

AssertEquals(
    Expected := expected,
    Actual := out,
    Message := 'Did not produce the expected boolean value from JSON for a true value'
);

TEST_FINISHED();
END_METHOD

METHOD PUBLIC TestTryGetKeyByte
VAR
    jsonDeserializer : JsonDeserializer;
    json : STRING := '{"data":100}';
    out : BYTE;
	feedback : DeserializerFeedback;
    expected : BYTE := 100;
END_VAR
TEST('TestTryGetKeyByte');

jsonDeserializer.TryLoad(json);
jsonDeserializer.TryGetKeyByte('data', out, feedback);

AssertEquals(
    Expected := expected,
    Actual := out,
    Message := 'Did not produce the expected BYTE value from JSON'
);

TEST_FINISHED();
END_METHOD

METHOD PUBLIC TestTryGetKeyDateTime
VAR
    jsonDeserializer : JsonDeserializer;
    json : STRING := '{"data":"2023-12-30T15:20:00"}';
    out : DATE_AND_TIME;
	feedback : DeserializerFeedback;
    expected : DATE_AND_TIME := DT#2023-12-30-15:20:00;
END_VAR
TEST('TestTryGetKeyDateTime');

jsonDeserializer.TryLoad(json);
jsonDeserializer.TryGetKeyDateTime('data', out, feedback);

AssertEquals(
    Expected := expected,
    Actual := out,
    Message := 'Did not produce the expected DATE_AND_TIME value from JSON'
);

TEST_FINISHED();
END_METHOD

METHOD PUBLIC TestTryGetKeyDcTime
VAR
    jsonDeserializer : JsonDeserializer;
    json : STRING := '{"data":"2000-01-01T00:00:00.012345678"}';
    out : DCTIME;
	feedback : DeserializerFeedback;
    expected : DCTIME := 12345678;
END_VAR
TEST('TestTryGetKeyDcTime');

jsonDeserializer.TryLoad(json);
jsonDeserializer.TryGetKeyDcTime('data', out, feedback);

AssertEquals(
    Expected := expected,
    Actual := out,
    Message := 'Did not produce the expected DCTIME value from JSON string'
);

TEST_FINISHED();
END_METHOD

METHOD PUBLIC TestTryGetKeyDint
VAR
    jsonDeserializer : JsonDeserializer;
    json : STRING := '{"data":12345}';
    out : DINT;
	feedback : DeserializerFeedback;
    expected : DINT := 12345;
END_VAR
TEST('TestTryGetKeyDint');

jsonDeserializer.TryLoad(json);
jsonDeserializer.TryGetKeyDint('data', out, feedback);

AssertEquals(
    Expected := expected,
    Actual := out,
    Message := 'Did not produce the expected DINT value from JSON'
);

TEST_FINISHED();
END_METHOD

METHOD PUBLIC TestTryGetKeyDword
VAR
    jsonDeserializer : JsonDeserializer;
    json : STRING := '{"data":12345}';
    out : DWORD;
	feedback : DeserializerFeedback;
    expected : DWORD := 12345;
END_VAR
TEST('TestTryGetKeyDword');

jsonDeserializer.TryLoad(json);
jsonDeserializer.TryGetKeyDword('data', out, feedback);

AssertEquals(
    Expected := expected,
    Actual := out,
    Message := 'Did not produce the expected DWORD value from JSON'
);

TEST_FINISHED();
END_METHOD

METHOD PUBLIC TestTryGetKeyFileTime
VAR
    jsonDeserializer : JsonDeserializer;
    json : STRING := '{"data":"1601-01-01T00:00:01.2345678"}';
    out : FILETIME;
	feedback : DeserializerFeedback;
    expected : FILETIME := 12345678;
END_VAR
TEST('TestTryGetKeyFileTime');

jsonDeserializer.TryLoad(json);
jsonDeserializer.TryGetKeyFileTime('data', out, feedback);

AssertEquals(
    Expected := expected,
    Actual := out,
    Message := 'Did not produce the expected FILETIME value from JSON string'
);

TEST_FINISHED();
END_METHOD

METHOD PUBLIC TestTryGetKeyHexAsBytes
VAR
    jsonDeserializer : JsonDeserializer;
    json : STRING := '{"data":"baadf00d"}';
    out : ARRAY[0..3] OF BYTE;
	feedback : DeserializerFeedback;
    expected : ARRAY[0..3] OF BYTE := [16#BA, 16#AD, 16#F0, 16#0D];
END_VAR
TEST('TestTryGetKeyHexAsBytes');

jsonDeserializer.TryLoad(json);
jsonDeserializer.TryGetKeyHexAsBytes('data', ADR(out), SIZEOF(out), feedback);

AssertEquals(
    Expected := expected,
    Actual := out,
    Message := 'Did not produce the expected binary data from JSON hexadecimal string'
);

TEST_FINISHED();
END_METHOD

METHOD PUBLIC TestTryGetKeyInt
VAR
    jsonDeserializer : JsonDeserializer;
    json : STRING := '{"data":12345}';
    out : INT;
	feedback : DeserializerFeedback;
    expected : INT := 12345;
END_VAR
TEST('TestTryGetKeyInt');

jsonDeserializer.TryLoad(json);
jsonDeserializer.TryGetKeyInt('data', out, feedback);

AssertEquals(
    Expected := expected,
    Actual := out,
    Message := 'Did not produce the expected INT value from JSON'
);

TEST_FINISHED();
END_METHOD

METHOD PUBLIC TestTryGetKeyLint
VAR
    jsonDeserializer : JsonDeserializer;
    json : STRING := '{"data":9223372036854775807}';
    out : LINT;
	feedback : DeserializerFeedback;
    expected : LINT := 9223372036854775807;
END_VAR
TEST('TestTryGetKeyLint');

jsonDeserializer.TryLoad(json);
jsonDeserializer.TryGetKeyLint('data', out, feedback);

AssertEquals(
    Expected := expected,
    Actual := out,
    Message := 'Did not produce the expected LINT value from JSON'
);

TEST_FINISHED();
END_METHOD

METHOD PUBLIC TestTryGetKeyLreal
VAR
    jsonDeserializer : JsonDeserializer;
    json : STRING := '{"data":123456.789}';
    out : LREAL;
	feedback : DeserializerFeedback;
    expected : LREAL := 123456.789;
END_VAR
TEST('TestTryGetKeyLreal');

jsonDeserializer.TryLoad(json);
jsonDeserializer.TryGetKeyLreal('data', out, feedback);

AssertEquals(
    Expected := expected,
    Actual := out,
    Message := 'Did not produce the expected LREAL value from JSON'
);

TEST_FINISHED();
END_METHOD

METHOD PUBLIC TestTryGetKeyLtime
VAR
    jsonDeserializer : JsonDeserializer;
    json : STRING := '{"data":"LTIME#100d2h30m40s500ms600us700ns"}';
    out : LTIME;
	feedback : DeserializerFeedback;
    expected : LTIME := LTIME#100D2H30M40S500MS600US700NS;
END_VAR
TEST('TestTryGetKeyLtime');

jsonDeserializer.TryLoad(json);
jsonDeserializer.TryGetKeyLtime('data', out, feedback);

AssertEquals(
    Expected := expected,
    Actual := out,
    Message := 'Did not produce the expected LTIME value from JSON string'
);

TEST_FINISHED();
END_METHOD

METHOD PUBLIC TestTryGetKeyLword
VAR
    jsonDeserializer : JsonDeserializer;
    json : STRING := '{"data":9223372036854775807}';
    out : LWORD;
	feedback : DeserializerFeedback;
    expected : LWORD := 9223372036854775807;
END_VAR
TEST('TestTryGetKeyLword');

jsonDeserializer.TryLoad(json);
jsonDeserializer.TryGetKeyLword('data', out, feedback);

AssertEquals(
    Expected := expected,
    Actual := out,
    Message := 'Did not produce the expected LWORD value from JSON'
);

TEST_FINISHED();
END_METHOD

METHOD PUBLIC TestTryGetKeyReal
VAR
    jsonDeserializer : JsonDeserializer;
    json : STRING := '{"data":123.4}';
    out : REAL;
	feedback : DeserializerFeedback;
    expected : REAL := 123.4;
END_VAR
TEST('TestTryGetKeyReal');

jsonDeserializer.TryLoad(json);
jsonDeserializer.TryGetKeyReal('data', out, feedback);

AssertEquals(
    Expected := expected,
    Actual := out,
    Message := 'Did not produce the expected REAL value from JSON'
);

TEST_FINISHED();
END_METHOD

METHOD PUBLIC TestTryGetKeySint
VAR
    jsonDeserializer : JsonDeserializer;
    json : STRING := '{"data":123}';
    out : SINT;
	feedback : DeserializerFeedback;
    expected : SINT := 123;
END_VAR
TEST('TestTryGetKeySint');

jsonDeserializer.TryLoad(json);
jsonDeserializer.TryGetKeySint('data', out, feedback);

AssertEquals(
    Expected := expected,
    Actual := out,
    Message := 'Did not produce the expected SINT value from JSON'
);

TEST_FINISHED();
END_METHOD

METHOD PUBLIC TestTryGetKeyString
VAR
    jsonDeserializer : JsonDeserializer;
    json : STRING := '{"data":"foobar"}';
    out : STRING;
	feedback : DeserializerFeedback;
    expected : STRING := 'foobar';
END_VAR
TEST('TestTryGetKeyString');

jsonDeserializer.TryLoad(json);
jsonDeserializer.TryGetKeyString('data', out, feedback);

AssertEquals(
    Expected := expected,
    Actual := out,
    Message := 'Did not produce the expected STRING value from JSON'
);

TEST_FINISHED();
END_METHOD

METHOD PUBLIC TestTryGetKeyTime
VAR
    jsonDeserializer : JsonDeserializer;
    json : STRING := '{"data":"T#49d17h2m47s295ms"}';
    out : TIME;
	feedback : DeserializerFeedback;
    expected : TIME := T#49D17H2M47S295MS;
END_VAR
TEST('TestTryGetKeyTime');

jsonDeserializer.TryLoad(json);
jsonDeserializer.TryGetKeyTime('data', out, feedback);

AssertEquals(
    Expected := expected,
    Actual := out,
    Message := 'Did not produce the expected TIME value from JSON'
);

TEST_FINISHED();
END_METHOD

METHOD PUBLIC TestTryGetKeyTod
VAR
    jsonDeserializer : JsonDeserializer;
    json : STRING := '{"data":"TOD#23:01:23.456"}';
    out : TOD;
	feedback : DeserializerFeedback;
    expected : TOD := TOD#23:01:23.456;
END_VAR
TEST('TestTryGetKeyTod');

jsonDeserializer.TryLoad(json);
jsonDeserializer.TryGetKeyTod('data', out, feedback);

AssertEquals(
    Expected := expected,
    Actual := out,
    Message := 'Did not produce the expected TOD value from JSON'
);

TEST_FINISHED();
END_METHOD

METHOD PUBLIC TestTryGetKeyUdint
VAR
    jsonDeserializer : JsonDeserializer;
    json : STRING := '{"data":123456}';
    out : UDINT;
	feedback : DeserializerFeedback;
    expected : UDINT := 123456;
END_VAR
TEST('TestTryGetKeyUdint');

jsonDeserializer.TryLoad(json);
jsonDeserializer.TryGetKeyUdint('data', out, feedback);

AssertEquals(
    Expected := expected,
    Actual := out,
    Message := 'Did not produce the expected UDINT value from JSON'
);

TEST_FINISHED();
END_METHOD

